FUNCTION_BLOCK "BFT_Garlic"   // FB362, LAD
{ S7_Optimized_Access := 'TRUE' }
VERSION : 0.1
// stored: AutoNumber false, IsIECCheckEnabled false, IsRetainMemResEnabled false, MemoryReserve 100, SetENOAutomatically false, UDAEnableTagReadback false
   VAR_INPUT
      IN_FBAV_Inload : Bool;
      IN_FBAV_Outlet : Bool;
      IN_FBAV_Transfer : Bool;
      IN_FBAV_CIP_Tank : Bool;
      IN_FBAV_CIP_Line : Bool;
      IN_FBP_Inload : Bool;
      IN_FBP_Inload_SP : Real;
      IN_FBP_Transfer : Bool;
      IN_FBP_Transfer_SP : Real;
      IN_FBP_CIP : Bool;
      IN_FBP_CIP_Sp : Real;
      IN_LT01 : Real;
      "LCS Start" : Bool;
      "LCS Stop" : Bool;
      "LCS EMS" : Bool;
      IN_Dose_Run : Bool;
      IN_Dose_Held : Bool;
      IN_Dose_Complete : Bool;
      IN_Dose_Header_1 : Bool;
      IN_Dose_Header_2 : Bool;
      IN_Dose_Valve_Cmd : Bool;
      IN_Dose_Pump_Cmd : Bool;
      IN_Dose_Pump_Sp : Real;
      IN_Dose_LineOK : Bool;
      "Inload Busy" : Bool;
      "CIP Pulse" : Bool;
      "CIP Supply ON" : Bool;
      "CIP Req OK" : Bool;
      "CIP Complete" : Bool;
      "CIP Busy" : Bool;
   END_VAR
   VAR_OUTPUT
      Out_AV_Inload : Bool;
      Out_AV_Outlet : Bool;
      Out_AV_Transfer : Bool;
      Out_AV_CIP_Tank : Bool;
      Out_AV_CIP_Line : Bool;
      Out_P_Inload : Bool;
      Out_P_Inload_Sp : Real;
      Out_P_Transfer : Bool;
      Out_P_Transfer_Sp : Real;
      Out_P_CIP : Bool;
      Out_P_CIP_Sp : Real;
      Out_XA : Bool;
      Out_XA_Speed : Real;
      Out_CIP_Req : Bool;
      Out_CIP_LineOpen : Bool;
   END_VAR
   VAR
      Cmd : Struct
         Inload : Bool;
         Ready_for_Tranfer : Bool;
         CIP_Tank : Bool;
         CIP_Line : Bool;
         Agitator_SpeedMode : Bool;
         Agitator_Mode : Bool;
         Agitator_Man_OnOff : Bool;
      END_STRUCT;
   END_VAR
   VAR RETAIN
      Param : Struct
         SP_Level_LL : Real := 10.0;
         SP_Level_ML : Real := 80.0;
         SP_Level_HL : Real := 100.0;
         SP_Level_Agi_ON1 : Real := 20.0;
         SP_Level_Agi_OFF1 : Real := 60.0;
         SP_Level_Agi_ON2 : Real := 62.0;
         SP_Level_Agi_OFF2 : Real := 80.0;
         SP_Level_Agi_ON3 : Real := 82.0;
         Agitator_SP_Speed : Real := 50.0;
         SupplyPump_SP_Speed : Real := 80.0;
         L_Hi_Lim : Real := 100.0;
         L_Lo_Lim : Real := 0.0;
         L_Hys : Real := 2.0;
         FlushingTime : DInt := 10000;
         CIP_Trf_SP_Speed : Real := 80.0;
         CIP_Ret_ON_SP : Real := 5.0;
         CIP_Ret_OFF_SP : Real;
      END_STRUCT;
   END_VAR
   VAR
      State : Struct   // Tank in loading state
         Tank_LL : Bool;
         Tank_ML : Bool;
         Tank_HL : Bool;
         Tank_inCIP : Bool;
         Tank_CIP_Enable : Bool;
         Line_inCIP : Bool;
         Line_CIP_Enable : Bool;
         CIP_Return_On : Bool;
         Inloading : Bool;
         Inload_Enable : Bool;
         Ready_For_Transfer : Bool;
         Ready_For_Transfer_Ena : Bool;
         Tank_Available : Bool;
         Transfer_On_Prog : Bool;
         L_Agi_ON1 : Bool;
         L_Agi_ON2 : Bool;
         L_Agi_ON3 : Bool;
      END_STRUCT;
      alwaysON : Bool;
      L_Hys_Abs : Real;
      Hys_Level_HL : Real;
      Hys_Level_ML : Real;
      Hys_Level_LL : Real;
      Hys_Level_Agi : Real;
      r : Struct
         PosE1 : Bool;
         PosE2 : Bool;
         PosE3 : Bool;
         PosE4 : Bool;
         PosE5 : Bool;
         PosE6 : Bool;
         PosE7 : Bool;
         PosE8 : Bool;
         PosE9 : Bool;
         PosE10 : Bool;
         PosE11 : Bool;
         PosE12 : Bool;
         PosE13 : Bool;
         PosE14 : Bool;
         PosE15 : Bool;
         PosE16 : Bool;
         PosE17 : Bool;
         PosE18 : Bool;
         PosE19 : Bool;
         PosE20 : Bool;
         PosE21 : Bool;
         PosE22 : Bool;
         PosE23 : Bool;
         PosE24 : Bool;
         PosE25 : Bool;
         PosE26 : Bool;
         PosE27 : Bool;
         PosE28 : Bool;
         PosE29 : Bool;
         PosE30 : Bool;
         PosE31 : Bool;
         PosE32 : Bool;
      END_STRUCT;
      Actuator : Struct
         AV_Inload : Bool;
         AV_Outlet : Bool;
         AV_Transfer : Bool;
         AV_CIP_Tank : Bool;
         AV_CIP_Line : Bool;
         P_Transfer : Bool;
         P_Inload : Bool;
         P_CIP : Bool;
         Agitator_level : Bool;
         LCS_OnOff : Bool;
      END_STRUCT;
      FlushingTim : TON_TIME;
      SPumpTim { S7_SetPoint := 'True'} : TON_TIME;
      AVinloadTim { S7_SetPoint := 'True'} : TON_TIME;
      L_AgiTim { S7_SetPoint := 'True'} : TON_TIME;
      Pump_TF_On_Time { S7_SetPoint := 'True'} : TON_TIME;
   END_VAR
   VAR_TEMP   // added for the SCL form of the ladder/FBD networks
      _w1 : Bool;
      _w2 : Bool;
   END_VAR
BEGIN

REGION Network 1: Always_ON
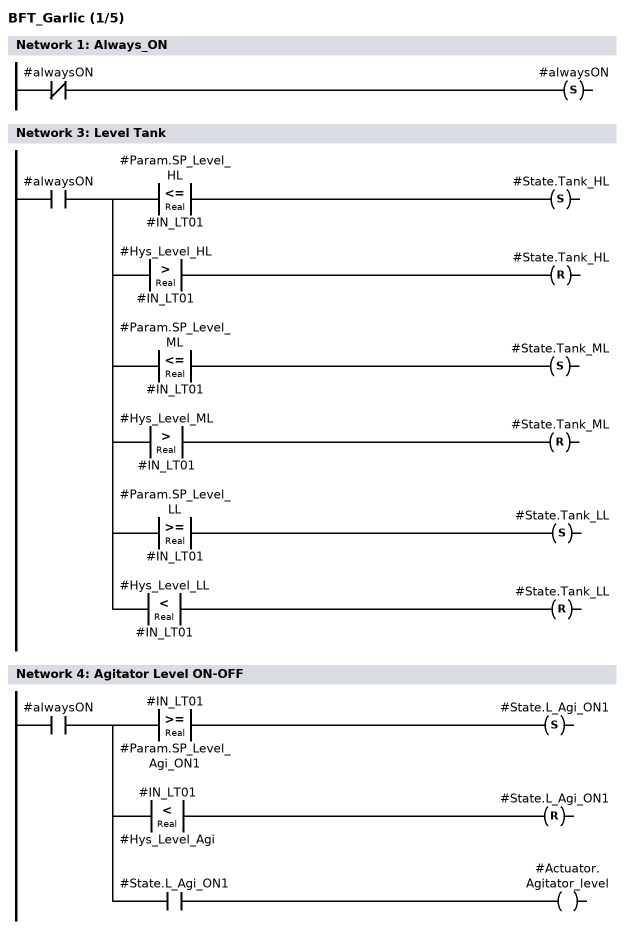
   RUNG wire#powerrail
      I_Contact( #alwaysON )
      S_Coil( #alwaysON )
   END_RUNG
   // the same network as SCL:
   IF NOT #alwaysON THEN #alwaysON := TRUE; END_IF;
END_REGION

NETWORK
TITLE = Hys Calculation
//Level Hys Absolute
      L     #Param.L_Hi_Lim;
      L     #Param.L_Lo_Lim;
      -R;
      L     100.0;
      /R;
      L     #Param.L_Hys;
      *R;
      T     #L_Hys_Abs;
//Tank High Level
      L     #Param.SP_Level_HL;
      L     #L_Hys_Abs;
      -R;
      T     #Hys_Level_HL;
//Tank Mid Level
      L     #Param.SP_Level_ML;
      L     #L_Hys_Abs;
      -R;
      T     #Hys_Level_ML;
//Tank Low Level
      L     #Param.SP_Level_LL;
      L     #L_Hys_Abs;
      +R;
      T     #Hys_Level_LL;
//Level Agi
      L     #Param.SP_Level_Agi_ON1;
      L     #L_Hys_Abs;
      -R;
      T     #Hys_Level_Agi;



REGION Network 3: Level Tank
   RUNG wire#powerrail
      Contact( #alwaysON )
      wire#w1
      { S7_Templates := "SrcType := Real" } LE_Contact(in1 := #Param.SP_Level_HL, in2 := #IN_LT01)
      S_Coil( #State.Tank_HL )
   END_RUNG
   RUNG wire#w1
      { S7_Templates := "SrcType := Real" } GT_Contact(in1 := #Hys_Level_HL, in2 := #IN_LT01)
      R_Coil( #State.Tank_HL )
   END_RUNG
   RUNG wire#w1
      { S7_Templates := "SrcType := Real" } LE_Contact(in1 := #Param.SP_Level_ML, in2 := #IN_LT01)
      S_Coil( #State.Tank_ML )
   END_RUNG
   RUNG wire#w1
      { S7_Templates := "SrcType := Real" } GT_Contact(in1 := #Hys_Level_ML, in2 := #IN_LT01)
      R_Coil( #State.Tank_ML )
   END_RUNG
   RUNG wire#w1
      { S7_Templates := "SrcType := Real" } GE_Contact(in1 := #Param.SP_Level_LL, in2 := #IN_LT01)
      S_Coil( #State.Tank_LL )
   END_RUNG
   RUNG wire#w1
      { S7_Templates := "SrcType := Real" } LT_Contact(in1 := #Hys_Level_LL, in2 := #IN_LT01)
      R_Coil( #State.Tank_LL )
   END_RUNG
   // the same network as SCL:
   IF #alwaysON AND (#Param.SP_Level_HL <= #IN_LT01) THEN #State.Tank_HL := TRUE; END_IF;
   IF #alwaysON AND (#Hys_Level_HL > #IN_LT01) THEN #State.Tank_HL := FALSE; END_IF;
   IF #alwaysON AND (#Param.SP_Level_ML <= #IN_LT01) THEN #State.Tank_ML := TRUE; END_IF;
   IF #alwaysON AND (#Hys_Level_ML > #IN_LT01) THEN #State.Tank_ML := FALSE; END_IF;
   IF #alwaysON AND (#Param.SP_Level_LL >= #IN_LT01) THEN #State.Tank_LL := TRUE; END_IF;
   IF #alwaysON AND (#Hys_Level_LL < #IN_LT01) THEN #State.Tank_LL := FALSE; END_IF;
END_REGION

REGION Network 4: Agitator Level ON-OFF
   RUNG wire#powerrail
      Contact( #alwaysON )
      wire#w1
      { S7_Templates := "SrcType := Real" } GE_Contact(in1 := #IN_LT01, in2 := #Param.SP_Level_Agi_ON1)
      S_Coil( #State.L_Agi_ON1 )
   END_RUNG
   RUNG wire#w1
      { S7_Templates := "SrcType := Real" } LT_Contact(in1 := #IN_LT01, in2 := #Hys_Level_Agi)
      R_Coil( #State.L_Agi_ON1 )
   END_RUNG
   RUNG wire#w1
      Contact( #State.L_Agi_ON1 )
      Coil( #Actuator.Agitator_level )
   END_RUNG
   // the same network as SCL:
   IF #alwaysON AND (#IN_LT01 >= #Param.SP_Level_Agi_ON1) THEN #State.L_Agi_ON1 := TRUE; END_IF;
   IF #alwaysON AND (#IN_LT01 < #Hys_Level_Agi) THEN #State.L_Agi_ON1 := FALSE; END_IF;
   #Actuator.Agitator_level := #alwaysON AND #State.L_Agi_ON1;
END_REGION

REGION Network 5: Agitator
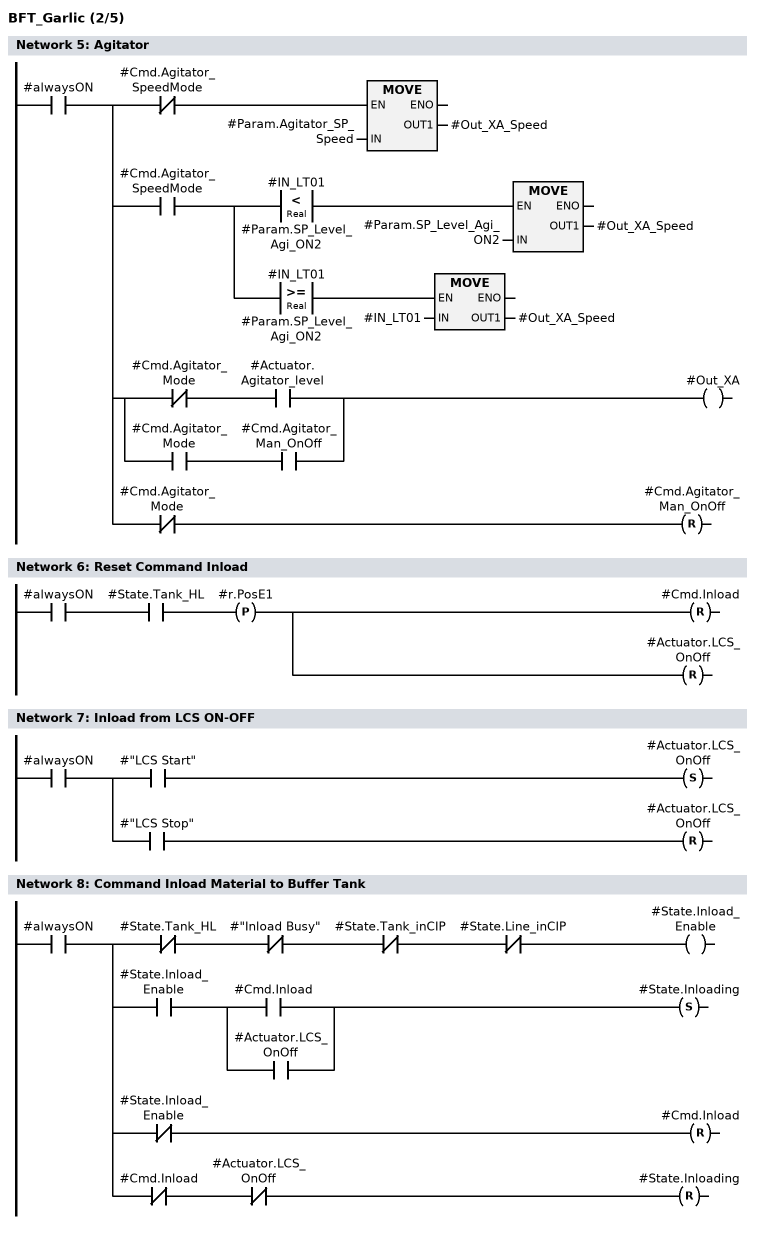
   RUNG wire#powerrail
      Contact( #alwaysON )
      wire#w1
      I_Contact( #Cmd.Agitator_SpeedMode )
      Move(in := #Param.Agitator_SP_Speed, out1 => #Out_XA_Speed)
   END_RUNG
   RUNG wire#w1
      Contact( #Cmd.Agitator_SpeedMode )
      wire#w2
      { S7_Templates := "SrcType := Real" } LT_Contact(in1 := #IN_LT01, in2 := #Param.SP_Level_Agi_ON2)
      Move(in := #Param.SP_Level_Agi_ON2, out1 => #Out_XA_Speed)
   END_RUNG
   RUNG wire#w2
      { S7_Templates := "SrcType := Real" } GE_Contact(in1 := #IN_LT01, in2 := #Param.SP_Level_Agi_ON2)
      Move(in := #IN_LT01, out1 => #Out_XA_Speed)
   END_RUNG
   RUNG wire#w1
      I_Contact( #Cmd.Agitator_Mode )
      Contact( #Actuator.Agitator_level )
      wire#w3
      Coil( #Out_XA )
   END_RUNG
   RUNG wire#w1
      Contact( #Cmd.Agitator_Mode )
      Contact( #Cmd.Agitator_Man_OnOff )
   END_RUNG wire#w3
   RUNG wire#w1
      I_Contact( #Cmd.Agitator_Mode )
      R_Coil( #Cmd.Agitator_Man_OnOff )
   END_RUNG
   // the same network as SCL:
   IF #alwaysON AND NOT #Cmd.Agitator_SpeedMode THEN #Out_XA_Speed := #Param.Agitator_SP_Speed; END_IF;
   #_w1 := #alwaysON AND #Cmd.Agitator_SpeedMode;
   IF #_w1 AND (#IN_LT01 < #Param.SP_Level_Agi_ON2) THEN #Out_XA_Speed := #Param.SP_Level_Agi_ON2; END_IF;
   IF #_w1 AND (#IN_LT01 >= #Param.SP_Level_Agi_ON2) THEN #Out_XA_Speed := #IN_LT01; END_IF;
   #Out_XA := #alwaysON AND ((NOT #Cmd.Agitator_Mode AND #Actuator.Agitator_level) OR (#Cmd.Agitator_Mode AND #Cmd.Agitator_Man_OnOff));
   IF #alwaysON AND NOT #Cmd.Agitator_Mode THEN #Cmd.Agitator_Man_OnOff := FALSE; END_IF;
END_REGION

REGION Network 6: Reset Command Inload
   RUNG wire#powerrail
      Contact( #alwaysON )
      Contact( #State.Tank_HL )
      P_Trig( #r.PosE1 )
      wire#w1
      R_Coil( #Cmd.Inload )
   END_RUNG
   RUNG wire#w1
      R_Coil( #Actuator.LCS_OnOff )
   END_RUNG
   // the same network as SCL:
   #_w1 := #alwaysON AND #State.Tank_HL;
   #_w2 := #_w1 AND NOT #r.PosE1;   // rising edge
   #r.PosE1 := #_w1;
   IF #_w2 THEN
       #Cmd.Inload := FALSE;
       #Actuator.LCS_OnOff := FALSE;
   END_IF;
END_REGION

REGION Network 7: Inload from LCS ON-OFF
   RUNG wire#powerrail
      Contact( #alwaysON )
      wire#w1
      Contact( #"LCS Start" )
      S_Coil( #Actuator.LCS_OnOff )
   END_RUNG
   RUNG wire#w1
      Contact( #"LCS Stop" )
      R_Coil( #Actuator.LCS_OnOff )
   END_RUNG
   // the same network as SCL:
   IF #alwaysON AND #"LCS Start" THEN #Actuator.LCS_OnOff := TRUE; END_IF;
   IF #alwaysON AND #"LCS Stop" THEN #Actuator.LCS_OnOff := FALSE; END_IF;
END_REGION

REGION Network 8: Command Inload Material to Buffer Tank
   RUNG wire#powerrail
      Contact( #alwaysON )
      wire#w1
      I_Contact( #State.Tank_HL )
      I_Contact( #"Inload Busy" )
      I_Contact( #State.Tank_inCIP )
      I_Contact( #State.Line_inCIP )
      Coil( #State.Inload_Enable )
   END_RUNG
   RUNG wire#w1
      Contact( #State.Inload_Enable )
      wire#w2
      Contact( #Cmd.Inload )
      wire#w3
      S_Coil( #State.Inloading )
   END_RUNG
   RUNG wire#w2
      Contact( #Actuator.LCS_OnOff )
   END_RUNG wire#w3
   RUNG wire#w1
      I_Contact( #State.Inload_Enable )
      R_Coil( #Cmd.Inload )
   END_RUNG
   RUNG wire#w1
      I_Contact( #Cmd.Inload )
      I_Contact( #Actuator.LCS_OnOff )
      R_Coil( #State.Inloading )
   END_RUNG
   // the same network as SCL:
   #State.Inload_Enable := #alwaysON AND NOT #State.Tank_HL AND NOT #"Inload Busy" AND NOT #State.Tank_inCIP AND NOT #State.Line_inCIP;
   IF #alwaysON AND #State.Inload_Enable AND (#Cmd.Inload OR #Actuator.LCS_OnOff) THEN
       #State.Inloading := TRUE;
   END_IF;
   IF #alwaysON AND NOT #State.Inload_Enable THEN #Cmd.Inload := FALSE; END_IF;
   IF #alwaysON AND NOT #Cmd.Inload AND NOT #Actuator.LCS_OnOff THEN #State.Inloading := FALSE; END_IF;
END_REGION

REGION Network 9: Tank Ready for Transfer to Blending
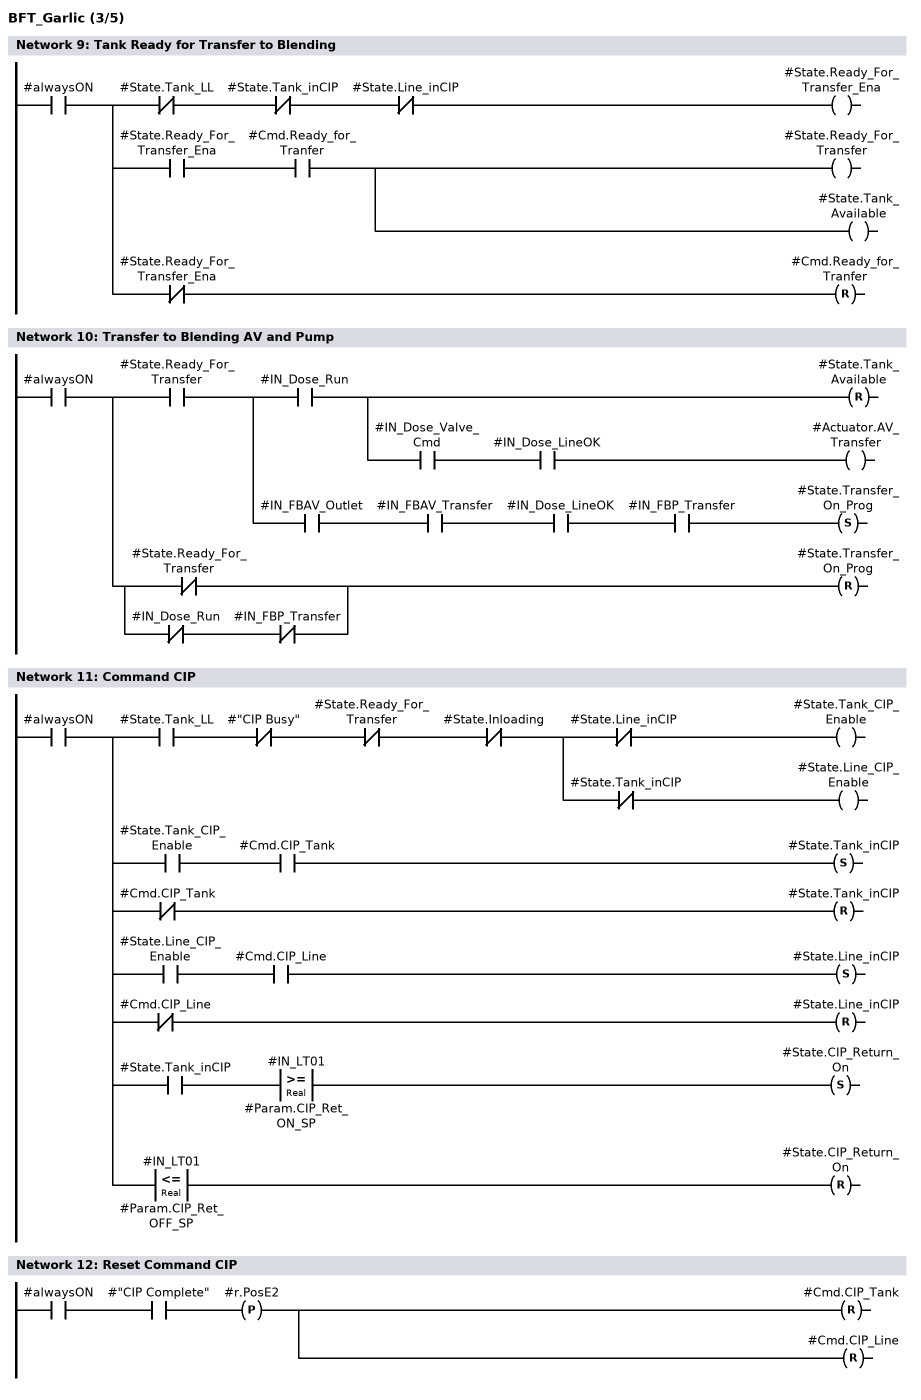
   RUNG wire#powerrail
      Contact( #alwaysON )
      wire#w1
      I_Contact( #State.Tank_LL )
      I_Contact( #State.Tank_inCIP )
      I_Contact( #State.Line_inCIP )
      Coil( #State.Ready_For_Transfer_Ena )
   END_RUNG
   RUNG wire#w1
      Contact( #State.Ready_For_Transfer_Ena )
      Contact( #Cmd.Ready_for_Tranfer )
      wire#w2
      Coil( #State.Ready_For_Transfer )
   END_RUNG
   RUNG wire#w2
      Coil( #State.Tank_Available )
   END_RUNG
   RUNG wire#w1
      I_Contact( #State.Ready_For_Transfer_Ena )
      R_Coil( #Cmd.Ready_for_Tranfer )
   END_RUNG
   // the same network as SCL:
   #State.Ready_For_Transfer_Ena := #alwaysON AND NOT #State.Tank_LL AND NOT #State.Tank_inCIP AND NOT #State.Line_inCIP;
   #State.Ready_For_Transfer := #alwaysON AND #State.Ready_For_Transfer_Ena AND #Cmd.Ready_for_Tranfer;
   #State.Tank_Available := #State.Ready_For_Transfer;
   IF #alwaysON AND NOT #State.Ready_For_Transfer_Ena THEN #Cmd.Ready_for_Tranfer := FALSE; END_IF;
END_REGION

REGION Network 10: Transfer to Blending AV and Pump
   RUNG wire#powerrail
      Contact( #alwaysON )
      wire#w1
      Contact( #State.Ready_For_Transfer )
      wire#w2
      Contact( #IN_Dose_Run )
      wire#w3
      R_Coil( #State.Tank_Available )
   END_RUNG
   RUNG wire#w3
      Contact( #IN_Dose_Valve_Cmd )
      Contact( #IN_Dose_LineOK )
      Coil( #Actuator.AV_Transfer )
   END_RUNG
   RUNG wire#w2
      Contact( #IN_FBAV_Outlet )
      Contact( #IN_FBAV_Transfer )
      Contact( #IN_Dose_LineOK )
      Contact( #IN_FBP_Transfer )
      S_Coil( #State.Transfer_On_Prog )
   END_RUNG
   RUNG wire#w1
      I_Contact( #State.Ready_For_Transfer )
      wire#w4
      R_Coil( #State.Transfer_On_Prog )
   END_RUNG
   RUNG wire#w1
      I_Contact( #IN_Dose_Run )
      I_Contact( #IN_FBP_Transfer )
   END_RUNG wire#w4
   // the same network as SCL:
   #_w1 := #alwaysON AND #State.Ready_For_Transfer;
   #_w2 := #_w1 AND #IN_Dose_Run;
   IF #_w2 THEN #State.Tank_Available := FALSE; END_IF;
   #Actuator.AV_Transfer := #_w2 AND #IN_Dose_Valve_Cmd AND #IN_Dose_LineOK;
   IF #_w1 AND #IN_FBAV_Outlet AND #IN_FBAV_Transfer AND #IN_Dose_LineOK AND #IN_FBP_Transfer THEN
       #State.Transfer_On_Prog := TRUE;
   END_IF;
   IF #alwaysON AND (NOT #State.Ready_For_Transfer OR (NOT #IN_Dose_Run AND NOT #IN_FBP_Transfer)) THEN
       #State.Transfer_On_Prog := FALSE;
   END_IF;
END_REGION

REGION Network 11: Command CIP
   RUNG wire#powerrail
      Contact( #alwaysON )
      wire#w1
      Contact( #State.Tank_LL )
      I_Contact( #"CIP Busy" )
      I_Contact( #State.Ready_For_Transfer )
      I_Contact( #State.Inloading )
      wire#w2
      I_Contact( #State.Line_inCIP )
      Coil( #State.Tank_CIP_Enable )
   END_RUNG
   RUNG wire#w2
      I_Contact( #State.Tank_inCIP )
      Coil( #State.Line_CIP_Enable )
   END_RUNG
   RUNG wire#w1
      Contact( #State.Tank_CIP_Enable )
      Contact( #Cmd.CIP_Tank )
      S_Coil( #State.Tank_inCIP )
   END_RUNG
   RUNG wire#w1
      I_Contact( #Cmd.CIP_Tank )
      R_Coil( #State.Tank_inCIP )
   END_RUNG
   RUNG wire#w1
      Contact( #State.Line_CIP_Enable )
      Contact( #Cmd.CIP_Line )
      S_Coil( #State.Line_inCIP )
   END_RUNG
   RUNG wire#w1
      I_Contact( #Cmd.CIP_Line )
      R_Coil( #State.Line_inCIP )
   END_RUNG
   RUNG wire#w1
      Contact( #State.Tank_inCIP )
      { S7_Templates := "SrcType := Real" } GE_Contact(in1 := #IN_LT01, in2 := #Param.CIP_Ret_ON_SP)
      S_Coil( #State.CIP_Return_On )
   END_RUNG
   RUNG wire#w1
      { S7_Templates := "SrcType := Real" } LE_Contact(in1 := #IN_LT01, in2 := #Param.CIP_Ret_OFF_SP)
      R_Coil( #State.CIP_Return_On )
   END_RUNG
   // the same network as SCL:
   #_w1 := #alwaysON AND #State.Tank_LL AND NOT #"CIP Busy" AND NOT #State.Ready_For_Transfer AND NOT #State.Inloading;
   #State.Tank_CIP_Enable := #_w1 AND NOT #State.Line_inCIP;
   #State.Line_CIP_Enable := #_w1 AND NOT #State.Tank_inCIP;
   IF #alwaysON AND #State.Tank_CIP_Enable AND #Cmd.CIP_Tank THEN #State.Tank_inCIP := TRUE; END_IF;
   IF #alwaysON AND NOT #Cmd.CIP_Tank THEN #State.Tank_inCIP := FALSE; END_IF;
   IF #alwaysON AND #State.Line_CIP_Enable AND #Cmd.CIP_Line THEN #State.Line_inCIP := TRUE; END_IF;
   IF #alwaysON AND NOT #Cmd.CIP_Line THEN #State.Line_inCIP := FALSE; END_IF;
   IF #alwaysON AND #State.Tank_inCIP AND (#IN_LT01 >= #Param.CIP_Ret_ON_SP) THEN
       #State.CIP_Return_On := TRUE;
   END_IF;
   IF #alwaysON AND (#IN_LT01 <= #Param.CIP_Ret_OFF_SP) THEN #State.CIP_Return_On := FALSE; END_IF;
END_REGION

REGION Network 12: Reset Command CIP
   RUNG wire#powerrail
      Contact( #alwaysON )
      Contact( #"CIP Complete" )
      P_Trig( #r.PosE2 )
      wire#w1
      R_Coil( #Cmd.CIP_Tank )
   END_RUNG
   RUNG wire#w1
      R_Coil( #Cmd.CIP_Line )
   END_RUNG
   // the same network as SCL:
   #_w1 := #alwaysON AND #"CIP Complete";
   #_w2 := #_w1 AND NOT #r.PosE2;   // rising edge
   #r.PosE2 := #_w1;
   IF #_w2 THEN
       #Cmd.CIP_Tank := FALSE;
       #Cmd.CIP_Line := FALSE;
   END_IF;
END_REGION

REGION Network 13: CIP Request and CIP Line Open
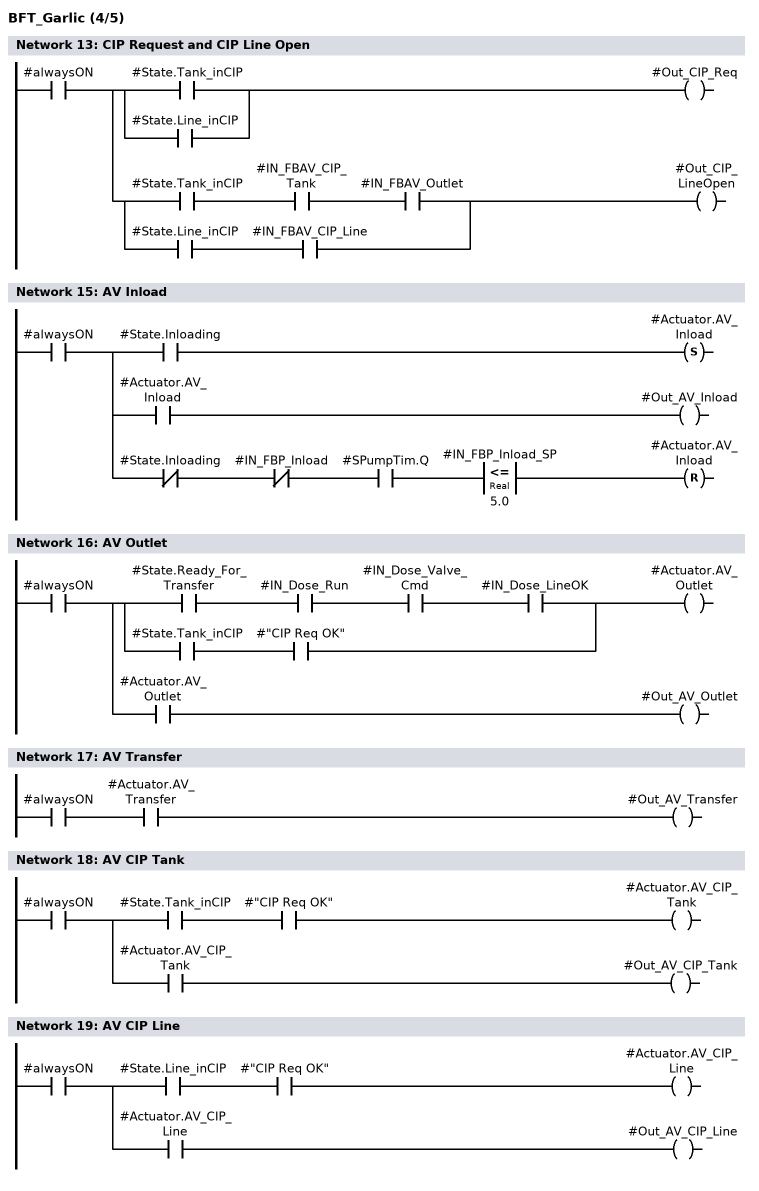
   RUNG wire#powerrail
      Contact( #alwaysON )
      wire#w1
      Contact( #State.Tank_inCIP )
      wire#w2
      Coil( #Out_CIP_Req )
   END_RUNG
   RUNG wire#w1
      Contact( #State.Line_inCIP )
   END_RUNG wire#w2
   RUNG wire#w1
      Contact( #State.Tank_inCIP )
      Contact( #IN_FBAV_CIP_Tank )
      Contact( #IN_FBAV_Outlet )
      wire#w3
      Coil( #Out_CIP_LineOpen )
   END_RUNG
   RUNG wire#w1
      Contact( #State.Line_inCIP )
      Contact( #IN_FBAV_CIP_Line )
   END_RUNG wire#w3
   // the same network as SCL:
   #Out_CIP_Req := #alwaysON AND (#State.Tank_inCIP OR #State.Line_inCIP);
   #Out_CIP_LineOpen := #alwaysON AND ((#State.Tank_inCIP AND #IN_FBAV_CIP_Tank AND #IN_FBAV_Outlet) OR (#State.Line_inCIP AND #IN_FBAV_CIP_Line));
END_REGION

REGION Network 15: AV Inload
   RUNG wire#powerrail
      Contact( #alwaysON )
      wire#w1
      Contact( #State.Inloading )
      S_Coil( #Actuator.AV_Inload )
   END_RUNG
   RUNG wire#w1
      Contact( #Actuator.AV_Inload )
      Coil( #Out_AV_Inload )
   END_RUNG
   RUNG wire#w1
      I_Contact( #State.Inloading )
      I_Contact( #IN_FBP_Inload )
      Contact( #SPumpTim.Q )
      { S7_Templates := "SrcType := Real" } LE_Contact(in1 := #IN_FBP_Inload_SP, in2 := 5.0)
      R_Coil( #Actuator.AV_Inload )
   END_RUNG
   // the same network as SCL:
   IF #alwaysON AND #State.Inloading THEN #Actuator.AV_Inload := TRUE; END_IF;
   #Out_AV_Inload := #alwaysON AND #Actuator.AV_Inload;
   IF #alwaysON AND NOT #State.Inloading AND NOT #IN_FBP_Inload AND #SPumpTim.Q AND (#IN_FBP_Inload_SP <= 5.0) THEN
       #Actuator.AV_Inload := FALSE;
   END_IF;
END_REGION

REGION Network 16: AV Outlet
   RUNG wire#powerrail
      Contact( #alwaysON )
      wire#w1
      Contact( #State.Ready_For_Transfer )
      Contact( #IN_Dose_Run )
      Contact( #IN_Dose_Valve_Cmd )
      Contact( #IN_Dose_LineOK )
      wire#w2
      Coil( #Actuator.AV_Outlet )
   END_RUNG
   RUNG wire#w1
      Contact( #State.Tank_inCIP )
      Contact( #"CIP Req OK" )
   END_RUNG wire#w2
   RUNG wire#w1
      Contact( #Actuator.AV_Outlet )
      Coil( #Out_AV_Outlet )
   END_RUNG
   // the same network as SCL:
   #Actuator.AV_Outlet := #alwaysON AND ((#State.Ready_For_Transfer AND #IN_Dose_Run AND #IN_Dose_Valve_Cmd AND #IN_Dose_LineOK) OR (#State.Tank_inCIP AND #"CIP Req OK"));
   #Out_AV_Outlet := #alwaysON AND #Actuator.AV_Outlet;
END_REGION

REGION Network 17: AV Transfer
   RUNG wire#powerrail
      Contact( #alwaysON )
      Contact( #Actuator.AV_Transfer )
      Coil( #Out_AV_Transfer )
   END_RUNG
   // the same network as SCL:
   #Out_AV_Transfer := #alwaysON AND #Actuator.AV_Transfer;
END_REGION

REGION Network 18: AV CIP Tank
   RUNG wire#powerrail
      Contact( #alwaysON )
      wire#w1
      Contact( #State.Tank_inCIP )
      Contact( #"CIP Req OK" )
      Coil( #Actuator.AV_CIP_Tank )
   END_RUNG
   RUNG wire#w1
      Contact( #Actuator.AV_CIP_Tank )
      Coil( #Out_AV_CIP_Tank )
   END_RUNG
   // the same network as SCL:
   #Actuator.AV_CIP_Tank := #alwaysON AND #State.Tank_inCIP AND #"CIP Req OK";
   #Out_AV_CIP_Tank := #alwaysON AND #Actuator.AV_CIP_Tank;
END_REGION

REGION Network 19: AV CIP Line
   RUNG wire#powerrail
      Contact( #alwaysON )
      wire#w1
      Contact( #State.Line_inCIP )
      Contact( #"CIP Req OK" )
      Coil( #Actuator.AV_CIP_Line )
   END_RUNG
   RUNG wire#w1
      Contact( #Actuator.AV_CIP_Line )
      Coil( #Out_AV_CIP_Line )
   END_RUNG
   // the same network as SCL:
   #Actuator.AV_CIP_Line := #alwaysON AND #State.Line_inCIP AND #"CIP Req OK";
   #Out_AV_CIP_Line := #alwaysON AND #Actuator.AV_CIP_Line;
END_REGION

REGION Network 21: Pump Inload
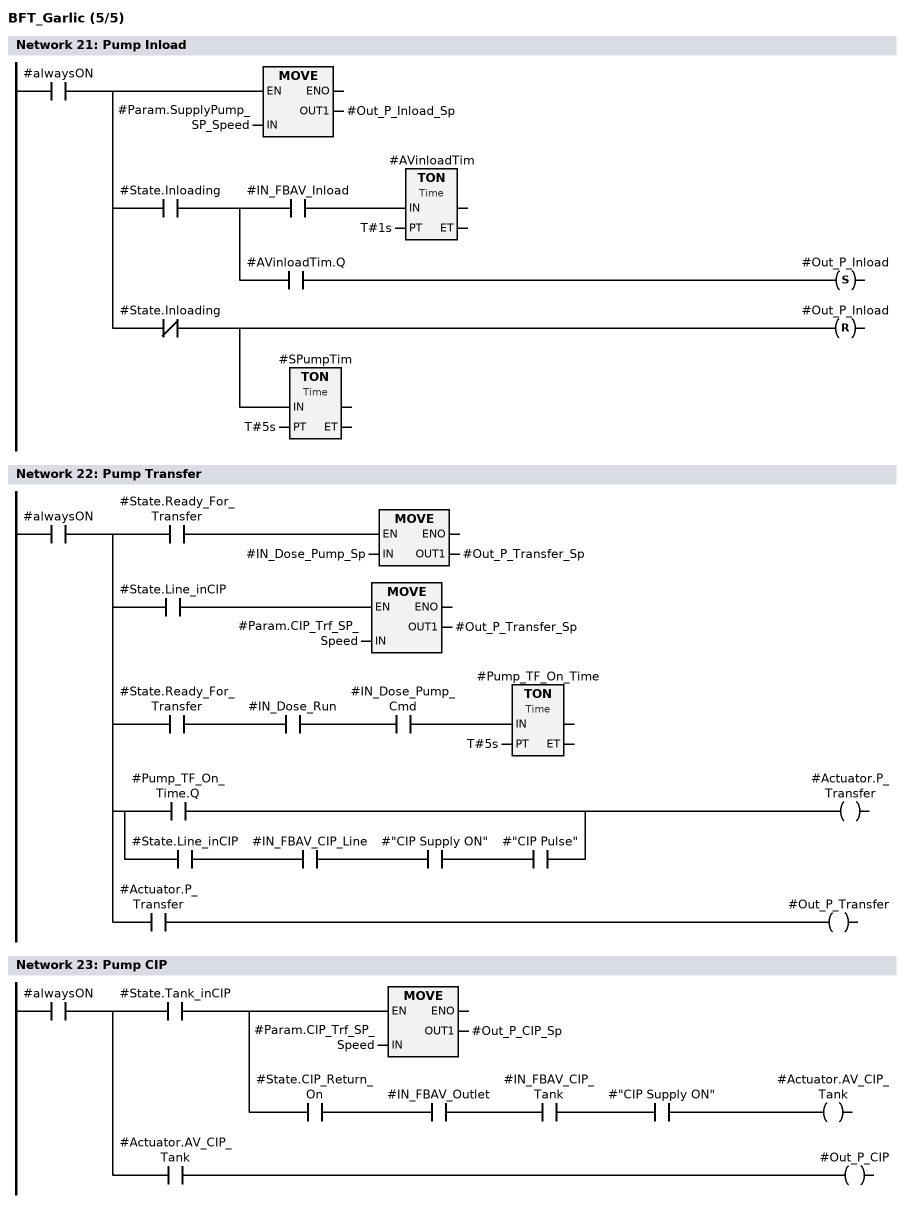
   RUNG wire#powerrail
      Contact( #alwaysON )
      wire#w1
      Move(in := #Param.SupplyPump_SP_Speed, out1 => #Out_P_Inload_Sp)
   END_RUNG
   RUNG wire#w1
      Contact( #State.Inloading )
      wire#w2
      Contact( #IN_FBAV_Inload )
      { S7_Templates := "time_type := Time" } #AVinloadTim.TON(pt := T#1s, et =>)
   END_RUNG
   RUNG wire#w2
      Contact( #AVinloadTim.Q )
      S_Coil( #Out_P_Inload )
   END_RUNG
   RUNG wire#w1
      I_Contact( #State.Inloading )
      wire#w3
      R_Coil( #Out_P_Inload )
   END_RUNG
   RUNG wire#w3
      { S7_Templates := "time_type := Time" } #SPumpTim.TON(pt := T#5s, et =>)
   END_RUNG
   // the same network as SCL:
   IF #alwaysON THEN #Out_P_Inload_Sp := #Param.SupplyPump_SP_Speed; END_IF;
   #_w1 := #alwaysON AND #State.Inloading;
   #AVinloadTim(IN := #_w1 AND #IN_FBAV_Inload, PT := T#1s);   // TON
   IF #_w1 AND #AVinloadTim.Q THEN #Out_P_Inload := TRUE; END_IF;
   #_w2 := #alwaysON AND NOT #State.Inloading;
   IF #_w2 THEN #Out_P_Inload := FALSE; END_IF;
   #SPumpTim(IN := #_w2, PT := T#5s);   // TON
END_REGION

REGION Network 22: Pump Transfer
   RUNG wire#powerrail
      Contact( #alwaysON )
      wire#w1
      Contact( #State.Ready_For_Transfer )
      Move(in := #IN_Dose_Pump_Sp, out1 => #Out_P_Transfer_Sp)
   END_RUNG
   RUNG wire#w1
      Contact( #State.Line_inCIP )
      Move(in := #Param.CIP_Trf_SP_Speed, out1 => #Out_P_Transfer_Sp)
   END_RUNG
   RUNG wire#w1
      Contact( #State.Ready_For_Transfer )
      Contact( #IN_Dose_Run )
      Contact( #IN_Dose_Pump_Cmd )
      { S7_Templates := "time_type := Time" } #Pump_TF_On_Time.TON(pt := T#5s, et =>)
   END_RUNG
   RUNG wire#w1
      Contact( #Pump_TF_On_Time.Q )
      wire#w2
      Coil( #Actuator.P_Transfer )
   END_RUNG
   RUNG wire#w1
      Contact( #State.Line_inCIP )
      Contact( #IN_FBAV_CIP_Line )
      Contact( #"CIP Supply ON" )
      Contact( #"CIP Pulse" )
   END_RUNG wire#w2
   RUNG wire#w1
      Contact( #Actuator.P_Transfer )
      Coil( #Out_P_Transfer )
   END_RUNG
   // the same network as SCL:
   IF #alwaysON AND #State.Ready_For_Transfer THEN #Out_P_Transfer_Sp := #IN_Dose_Pump_Sp; END_IF;
   IF #alwaysON AND #State.Line_inCIP THEN #Out_P_Transfer_Sp := #Param.CIP_Trf_SP_Speed; END_IF;
   #Pump_TF_On_Time(IN := #alwaysON AND #State.Ready_For_Transfer AND #IN_Dose_Run AND #IN_Dose_Pump_Cmd,   // TON
                    PT := T#5s);
   #Actuator.P_Transfer := #alwaysON AND (#Pump_TF_On_Time.Q OR (#State.Line_inCIP AND #IN_FBAV_CIP_Line AND #"CIP Supply ON" AND #"CIP Pulse"));
   #Out_P_Transfer := #alwaysON AND #Actuator.P_Transfer;
END_REGION

REGION Network 23: Pump CIP
   RUNG wire#powerrail
      Contact( #alwaysON )
      wire#w1
      Contact( #State.Tank_inCIP )
      wire#w2
      Move(in := #Param.CIP_Trf_SP_Speed, out1 => #Out_P_CIP_Sp)
   END_RUNG
   RUNG wire#w2
      Contact( #State.CIP_Return_On )
      Contact( #IN_FBAV_Outlet )
      Contact( #IN_FBAV_CIP_Tank )
      Contact( #"CIP Supply ON" )
      Coil( #Actuator.AV_CIP_Tank )
   END_RUNG
   RUNG wire#w1
      Contact( #Actuator.AV_CIP_Tank )
      Coil( #Out_P_CIP )
   END_RUNG
   // the same network as SCL:
   #_w1 := #alwaysON AND #State.Tank_inCIP;
   IF #_w1 THEN #Out_P_CIP_Sp := #Param.CIP_Trf_SP_Speed; END_IF;
   #Actuator.AV_CIP_Tank := #_w1 AND #State.CIP_Return_On AND #IN_FBAV_Outlet AND #IN_FBAV_CIP_Tank AND #"CIP Supply ON";
   #Out_P_CIP := #alwaysON AND #Actuator.AV_CIP_Tank;
END_REGION
END_FUNCTION_BLOCK

FUNCTION_BLOCK "BFT_Vinegar"   // FB363, LAD
{ S7_Optimized_Access := 'TRUE' }
VERSION : 0.1
// stored: AutoNumber false, IsIECCheckEnabled false, IsRetainMemResEnabled false, MemoryReserve 100, SetENOAutomatically false, UDAEnableTagReadback false
   VAR_INPUT
      IN_FBAV_Inload : Bool;
      IN_FBAV_Outlet : Bool;
      IN_FBAV_Transfer : Bool;
      IN_FBAV_CIP_Tank : Bool;
      IN_FBAV_CIP_Line : Bool;
      IN_FBP_Inload : Bool;
      IN_FBP_Inload_SP : Real;
      IN_FBP_Transfer : Bool;
      IN_FBP_Transfer_SP : Real;
      IN_FBP_CIP : Bool;
      IN_FBP_CIP_Sp : Real;
      IN_LT01 : Real;
      "LCS Start" : Bool;
      "LCS Stop" : Bool;
      "LCS EMS" : Bool;
      IN_Dose_Run : Bool;
      IN_Dose_Held : Bool;
      IN_Dose_Complete : Bool;
      IN_Dose_Valve_Cmd : Bool;
      IN_Dose_Pump_Cmd : Bool;
      IN_Dose_Pump_Sp : Real;
      IN_Dose_LineOK : Bool;
      "Inload Busy" : Bool;
      "CIP Pulse" : Bool;
      "CIP Supply ON" : Bool;
      "CIP Req OK" : Bool;
      "CIP Complete" : Bool;
      "CIP Busy" : Bool;
   END_VAR
   VAR_OUTPUT
      Out_AV_Inload : Bool;
      Out_AV_Outlet : Bool;
      Out_AV_Transfer : Bool;
      Out_AV_CIP_Tank : Bool;
      Out_AV_CIP_Line : Bool;
      Out_P_Inload : Bool;
      Out_P_Inload_Sp : Real;
      Out_P_Transfer : Bool;
      Out_P_Transfer_Sp : Real;
      Out_P_CIP : Bool;
      Out_P_CIP_Sp : Real;
      Out_CIP_Req : Bool;
      Out_CIP_LineOpen : Bool;
   END_VAR
   VAR
      Cmd : Struct
         Inload : Bool;
         Ready_for_Tranfer : Bool;
         CIP_Tank : Bool;
         CIP_Line : Bool;
      END_STRUCT;
   END_VAR
   VAR RETAIN
      Param : Struct
         SP_Level_LL : Real := 10.0;
         SP_Level_ML : Real := 80.0;
         SP_Level_HL : Real := 100.0;
         SupplyPump_SP_Speed : Real := 80.0;
         L_Hi_Lim : Real := 100.0;
         L_Lo_Lim : Real := 0.0;
         L_Hys : Real := 2.0;
         FlushingTime : DInt := 10000;
         CIP_Trf_SP_Speed : Real := 80.0;
         CIP_Ret_ON_SP : Real := 5.0;
         CIP_Ret_OFF_SP : Real;
      END_STRUCT;
   END_VAR
   VAR
      State : Struct   // Tank in loading state
         Tank_LL : Bool;
         Tank_ML : Bool;
         Tank_HL : Bool;
         Tank_inCIP : Bool;
         Tank_CIP_Enable : Bool;
         Line_inCIP : Bool;
         Line_CIP_Enable : Bool;
         CIP_Return_On : Bool;
         Inloading : Bool;
         Inload_Enable : Bool;
         Ready_For_Transfer : Bool;
         Ready_For_Transfer_Ena : Bool;
         Tank_Available : Bool;
         Transfer_On_Prog : Bool;
      END_STRUCT;
      alwaysON : Bool;
      L_Hys_Abs : Real;
      Hys_Level_HL : Real;
      Hys_Level_ML : Real;
      Hys_Level_LL : Real;
      r : Struct
         PosE1 : Bool;
         PosE2 : Bool;
         PosE3 : Bool;
         PosE4 : Bool;
         PosE5 : Bool;
         PosE6 : Bool;
         PosE7 : Bool;
         PosE8 : Bool;
         PosE9 : Bool;
         PosE10 : Bool;
         PosE11 : Bool;
         PosE12 : Bool;
         PosE13 : Bool;
         PosE14 : Bool;
         PosE15 : Bool;
         PosE16 : Bool;
         PosE17 : Bool;
         PosE18 : Bool;
         PosE19 : Bool;
         PosE20 : Bool;
         PosE21 : Bool;
         PosE22 : Bool;
         PosE23 : Bool;
         PosE24 : Bool;
         PosE25 : Bool;
         PosE26 : Bool;
         PosE27 : Bool;
         PosE28 : Bool;
         PosE29 : Bool;
         PosE30 : Bool;
         PosE31 : Bool;
         PosE32 : Bool;
      END_STRUCT;
      Actuator : Struct
         AV_Inload : Bool;
         AV_Outlet : Bool;
         AV_Transfer : Bool;
         AV_CIP_Tank : Bool;
         AV_CIP_Line : Bool;
         P_Transfer : Bool;
         P_Inload : Bool;
         P_CIP : Bool;
         LCS_OnOff : Bool;
      END_STRUCT;
      FlushingTim : TON_TIME;
      SPumpTim { S7_SetPoint := 'True'} : TON_TIME;
      AVinloadTim { S7_SetPoint := 'True'} : TON_TIME;
      Pump_TF_On_Time { S7_SetPoint := 'True'} : TON_TIME;
   END_VAR
   VAR_TEMP   // added for the SCL form of the ladder/FBD networks
      _w1 : Bool;
      _w2 : Bool;
   END_VAR
BEGIN

REGION Network 1: Always_ON
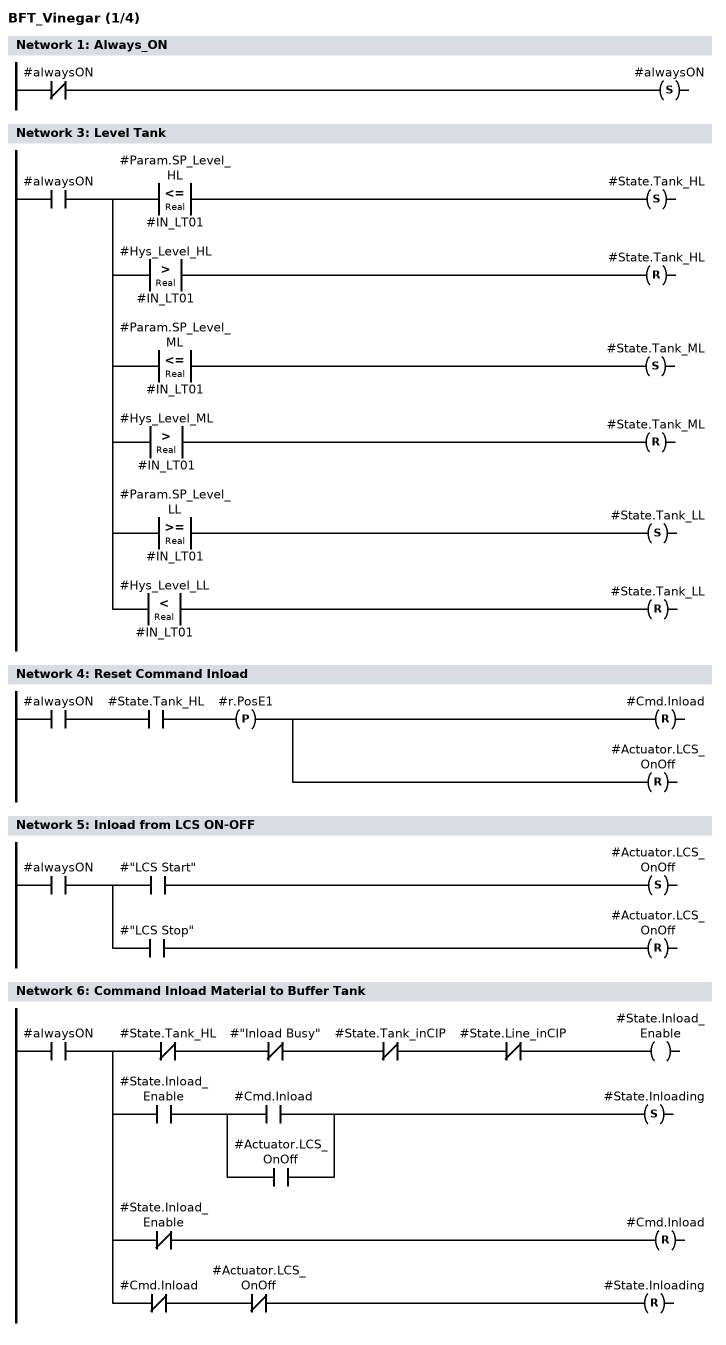
   RUNG wire#powerrail
      I_Contact( #alwaysON )
      S_Coil( #alwaysON )
   END_RUNG
   // the same network as SCL:
   IF NOT #alwaysON THEN #alwaysON := TRUE; END_IF;
END_REGION

NETWORK
TITLE = Hys Calculation
//Level Hys Absolute
      L     #Param.L_Hi_Lim;
      L     #Param.L_Lo_Lim;
      -R;
      L     100.0;
      /R;
      L     #Param.L_Hys;
      *R;
      T     #L_Hys_Abs;
//Tank High Level
      L     #Param.SP_Level_HL;
      L     #L_Hys_Abs;
      -R;
      T     #Hys_Level_HL;
//Tank Mid Level
      L     #Param.SP_Level_ML;
      L     #L_Hys_Abs;
      -R;
      T     #Hys_Level_ML;
//Tank Low Level
      L     #Param.SP_Level_LL;
      L     #L_Hys_Abs;
      +R;
      T     #Hys_Level_LL;


REGION Network 3: Level Tank
   RUNG wire#powerrail
      Contact( #alwaysON )
      wire#w1
      { S7_Templates := "SrcType := Real" } LE_Contact(in1 := #Param.SP_Level_HL, in2 := #IN_LT01)
      S_Coil( #State.Tank_HL )
   END_RUNG
   RUNG wire#w1
      { S7_Templates := "SrcType := Real" } GT_Contact(in1 := #Hys_Level_HL, in2 := #IN_LT01)
      R_Coil( #State.Tank_HL )
   END_RUNG
   RUNG wire#w1
      { S7_Templates := "SrcType := Real" } LE_Contact(in1 := #Param.SP_Level_ML, in2 := #IN_LT01)
      S_Coil( #State.Tank_ML )
   END_RUNG
   RUNG wire#w1
      { S7_Templates := "SrcType := Real" } GT_Contact(in1 := #Hys_Level_ML, in2 := #IN_LT01)
      R_Coil( #State.Tank_ML )
   END_RUNG
   RUNG wire#w1
      { S7_Templates := "SrcType := Real" } GE_Contact(in1 := #Param.SP_Level_LL, in2 := #IN_LT01)
      S_Coil( #State.Tank_LL )
   END_RUNG
   RUNG wire#w1
      { S7_Templates := "SrcType := Real" } LT_Contact(in1 := #Hys_Level_LL, in2 := #IN_LT01)
      R_Coil( #State.Tank_LL )
   END_RUNG
   // the same network as SCL:
   IF #alwaysON AND (#Param.SP_Level_HL <= #IN_LT01) THEN #State.Tank_HL := TRUE; END_IF;
   IF #alwaysON AND (#Hys_Level_HL > #IN_LT01) THEN #State.Tank_HL := FALSE; END_IF;
   IF #alwaysON AND (#Param.SP_Level_ML <= #IN_LT01) THEN #State.Tank_ML := TRUE; END_IF;
   IF #alwaysON AND (#Hys_Level_ML > #IN_LT01) THEN #State.Tank_ML := FALSE; END_IF;
   IF #alwaysON AND (#Param.SP_Level_LL >= #IN_LT01) THEN #State.Tank_LL := TRUE; END_IF;
   IF #alwaysON AND (#Hys_Level_LL < #IN_LT01) THEN #State.Tank_LL := FALSE; END_IF;
END_REGION

REGION Network 4: Reset Command Inload
   RUNG wire#powerrail
      Contact( #alwaysON )
      Contact( #State.Tank_HL )
      P_Trig( #r.PosE1 )
      wire#w1
      R_Coil( #Cmd.Inload )
   END_RUNG
   RUNG wire#w1
      R_Coil( #Actuator.LCS_OnOff )
   END_RUNG
   // the same network as SCL:
   #_w1 := #alwaysON AND #State.Tank_HL;
   #_w2 := #_w1 AND NOT #r.PosE1;   // rising edge
   #r.PosE1 := #_w1;
   IF #_w2 THEN
       #Cmd.Inload := FALSE;
       #Actuator.LCS_OnOff := FALSE;
   END_IF;
END_REGION

REGION Network 5: Inload from LCS ON-OFF
   RUNG wire#powerrail
      Contact( #alwaysON )
      wire#w1
      Contact( #"LCS Start" )
      S_Coil( #Actuator.LCS_OnOff )
   END_RUNG
   RUNG wire#w1
      Contact( #"LCS Stop" )
      R_Coil( #Actuator.LCS_OnOff )
   END_RUNG
   // the same network as SCL:
   IF #alwaysON AND #"LCS Start" THEN #Actuator.LCS_OnOff := TRUE; END_IF;
   IF #alwaysON AND #"LCS Stop" THEN #Actuator.LCS_OnOff := FALSE; END_IF;
END_REGION

REGION Network 6: Command Inload Material to Buffer Tank
   RUNG wire#powerrail
      Contact( #alwaysON )
      wire#w1
      I_Contact( #State.Tank_HL )
      I_Contact( #"Inload Busy" )
      I_Contact( #State.Tank_inCIP )
      I_Contact( #State.Line_inCIP )
      Coil( #State.Inload_Enable )
   END_RUNG
   RUNG wire#w1
      Contact( #State.Inload_Enable )
      wire#w2
      Contact( #Cmd.Inload )
      wire#w3
      S_Coil( #State.Inloading )
   END_RUNG
   RUNG wire#w2
      Contact( #Actuator.LCS_OnOff )
   END_RUNG wire#w3
   RUNG wire#w1
      I_Contact( #State.Inload_Enable )
      R_Coil( #Cmd.Inload )
   END_RUNG
   RUNG wire#w1
      I_Contact( #Cmd.Inload )
      I_Contact( #Actuator.LCS_OnOff )
      R_Coil( #State.Inloading )
   END_RUNG
   // the same network as SCL:
   #State.Inload_Enable := #alwaysON AND NOT #State.Tank_HL AND NOT #"Inload Busy" AND NOT #State.Tank_inCIP AND NOT #State.Line_inCIP;
   IF #alwaysON AND #State.Inload_Enable AND (#Cmd.Inload OR #Actuator.LCS_OnOff) THEN
       #State.Inloading := TRUE;
   END_IF;
   IF #alwaysON AND NOT #State.Inload_Enable THEN #Cmd.Inload := FALSE; END_IF;
   IF #alwaysON AND NOT #Cmd.Inload AND NOT #Actuator.LCS_OnOff THEN #State.Inloading := FALSE; END_IF;
END_REGION

REGION Network 7: Tank Ready for Transfer to Blending
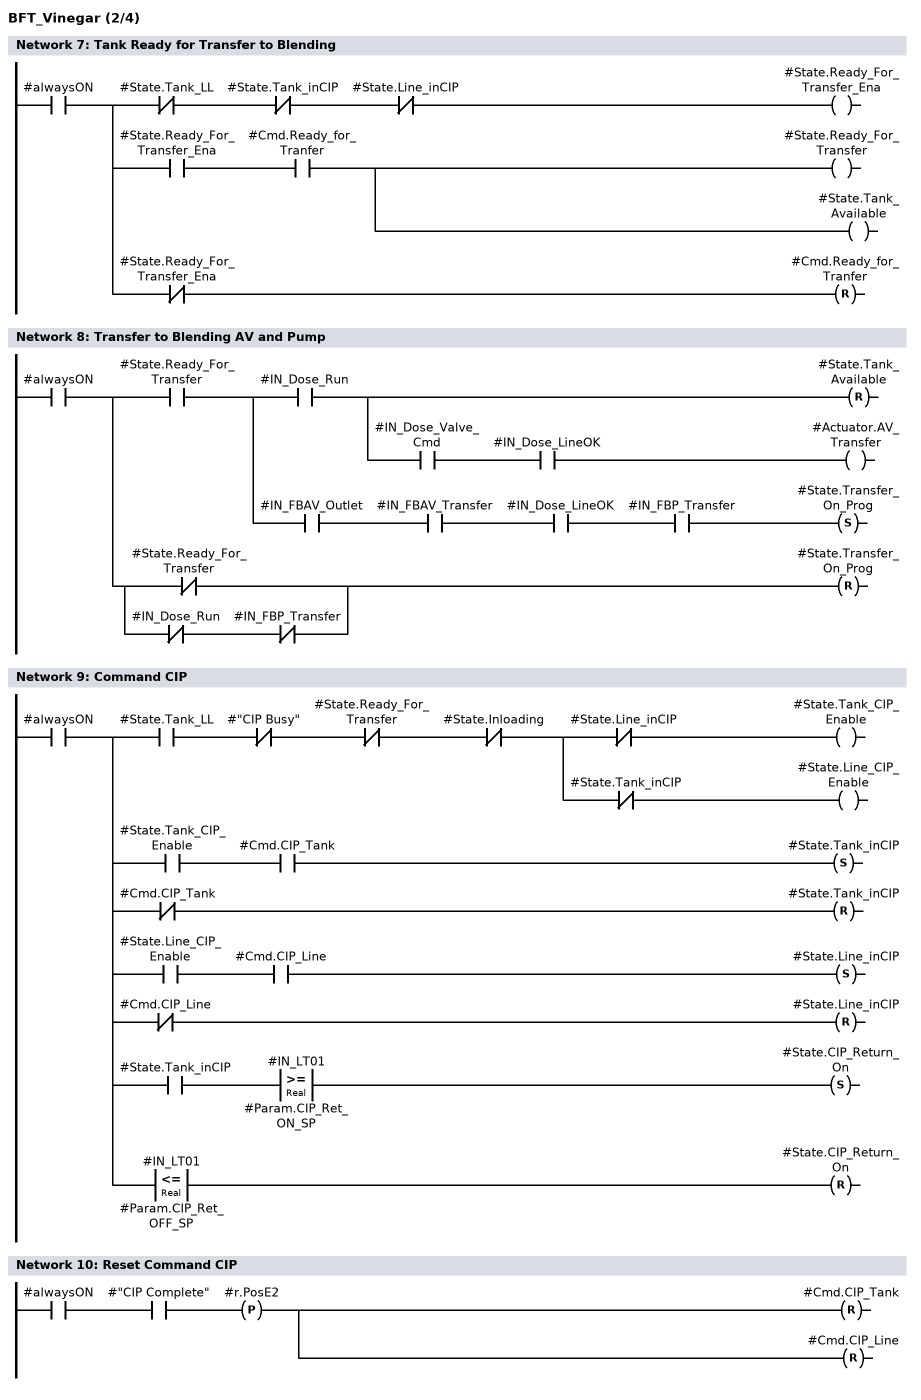
   RUNG wire#powerrail
      Contact( #alwaysON )
      wire#w1
      I_Contact( #State.Tank_LL )
      I_Contact( #State.Tank_inCIP )
      I_Contact( #State.Line_inCIP )
      Coil( #State.Ready_For_Transfer_Ena )
   END_RUNG
   RUNG wire#w1
      Contact( #State.Ready_For_Transfer_Ena )
      Contact( #Cmd.Ready_for_Tranfer )
      wire#w2
      Coil( #State.Ready_For_Transfer )
   END_RUNG
   RUNG wire#w2
      Coil( #State.Tank_Available )
   END_RUNG
   RUNG wire#w1
      I_Contact( #State.Ready_For_Transfer_Ena )
      R_Coil( #Cmd.Ready_for_Tranfer )
   END_RUNG
   // the same network as SCL:
   #State.Ready_For_Transfer_Ena := #alwaysON AND NOT #State.Tank_LL AND NOT #State.Tank_inCIP AND NOT #State.Line_inCIP;
   #State.Ready_For_Transfer := #alwaysON AND #State.Ready_For_Transfer_Ena AND #Cmd.Ready_for_Tranfer;
   #State.Tank_Available := #State.Ready_For_Transfer;
   IF #alwaysON AND NOT #State.Ready_For_Transfer_Ena THEN #Cmd.Ready_for_Tranfer := FALSE; END_IF;
END_REGION

REGION Network 8: Transfer to Blending AV and Pump
   RUNG wire#powerrail
      Contact( #alwaysON )
      wire#w1
      Contact( #State.Ready_For_Transfer )
      wire#w2
      Contact( #IN_Dose_Run )
      wire#w3
      R_Coil( #State.Tank_Available )
   END_RUNG
   RUNG wire#w3
      Contact( #IN_Dose_Valve_Cmd )
      Contact( #IN_Dose_LineOK )
      Coil( #Actuator.AV_Transfer )
   END_RUNG
   RUNG wire#w2
      Contact( #IN_FBAV_Outlet )
      Contact( #IN_FBAV_Transfer )
      Contact( #IN_Dose_LineOK )
      Contact( #IN_FBP_Transfer )
      S_Coil( #State.Transfer_On_Prog )
   END_RUNG
   RUNG wire#w1
      I_Contact( #State.Ready_For_Transfer )
      wire#w4
      R_Coil( #State.Transfer_On_Prog )
   END_RUNG
   RUNG wire#w1
      I_Contact( #IN_Dose_Run )
      I_Contact( #IN_FBP_Transfer )
   END_RUNG wire#w4
   // the same network as SCL:
   #_w1 := #alwaysON AND #State.Ready_For_Transfer;
   #_w2 := #_w1 AND #IN_Dose_Run;
   IF #_w2 THEN #State.Tank_Available := FALSE; END_IF;
   #Actuator.AV_Transfer := #_w2 AND #IN_Dose_Valve_Cmd AND #IN_Dose_LineOK;
   IF #_w1 AND #IN_FBAV_Outlet AND #IN_FBAV_Transfer AND #IN_Dose_LineOK AND #IN_FBP_Transfer THEN
       #State.Transfer_On_Prog := TRUE;
   END_IF;
   IF #alwaysON AND (NOT #State.Ready_For_Transfer OR (NOT #IN_Dose_Run AND NOT #IN_FBP_Transfer)) THEN
       #State.Transfer_On_Prog := FALSE;
   END_IF;
END_REGION

REGION Network 9: Command CIP
   RUNG wire#powerrail
      Contact( #alwaysON )
      wire#w1
      Contact( #State.Tank_LL )
      I_Contact( #"CIP Busy" )
      I_Contact( #State.Ready_For_Transfer )
      I_Contact( #State.Inloading )
      wire#w2
      I_Contact( #State.Line_inCIP )
      Coil( #State.Tank_CIP_Enable )
   END_RUNG
   RUNG wire#w2
      I_Contact( #State.Tank_inCIP )
      Coil( #State.Line_CIP_Enable )
   END_RUNG
   RUNG wire#w1
      Contact( #State.Tank_CIP_Enable )
      Contact( #Cmd.CIP_Tank )
      S_Coil( #State.Tank_inCIP )
   END_RUNG
   RUNG wire#w1
      I_Contact( #Cmd.CIP_Tank )
      R_Coil( #State.Tank_inCIP )
   END_RUNG
   RUNG wire#w1
      Contact( #State.Line_CIP_Enable )
      Contact( #Cmd.CIP_Line )
      S_Coil( #State.Line_inCIP )
   END_RUNG
   RUNG wire#w1
      I_Contact( #Cmd.CIP_Line )
      R_Coil( #State.Line_inCIP )
   END_RUNG
   RUNG wire#w1
      Contact( #State.Tank_inCIP )
      { S7_Templates := "SrcType := Real" } GE_Contact(in1 := #IN_LT01, in2 := #Param.CIP_Ret_ON_SP)
      S_Coil( #State.CIP_Return_On )
   END_RUNG
   RUNG wire#w1
      { S7_Templates := "SrcType := Real" } LE_Contact(in1 := #IN_LT01, in2 := #Param.CIP_Ret_OFF_SP)
      R_Coil( #State.CIP_Return_On )
   END_RUNG
   // the same network as SCL:
   #_w1 := #alwaysON AND #State.Tank_LL AND NOT #"CIP Busy" AND NOT #State.Ready_For_Transfer AND NOT #State.Inloading;
   #State.Tank_CIP_Enable := #_w1 AND NOT #State.Line_inCIP;
   #State.Line_CIP_Enable := #_w1 AND NOT #State.Tank_inCIP;
   IF #alwaysON AND #State.Tank_CIP_Enable AND #Cmd.CIP_Tank THEN #State.Tank_inCIP := TRUE; END_IF;
   IF #alwaysON AND NOT #Cmd.CIP_Tank THEN #State.Tank_inCIP := FALSE; END_IF;
   IF #alwaysON AND #State.Line_CIP_Enable AND #Cmd.CIP_Line THEN #State.Line_inCIP := TRUE; END_IF;
   IF #alwaysON AND NOT #Cmd.CIP_Line THEN #State.Line_inCIP := FALSE; END_IF;
   IF #alwaysON AND #State.Tank_inCIP AND (#IN_LT01 >= #Param.CIP_Ret_ON_SP) THEN
       #State.CIP_Return_On := TRUE;
   END_IF;
   IF #alwaysON AND (#IN_LT01 <= #Param.CIP_Ret_OFF_SP) THEN #State.CIP_Return_On := FALSE; END_IF;
END_REGION

REGION Network 10: Reset Command CIP
   RUNG wire#powerrail
      Contact( #alwaysON )
      Contact( #"CIP Complete" )
      P_Trig( #r.PosE2 )
      wire#w1
      R_Coil( #Cmd.CIP_Tank )
   END_RUNG
   RUNG wire#w1
      R_Coil( #Cmd.CIP_Line )
   END_RUNG
   // the same network as SCL:
   #_w1 := #alwaysON AND #"CIP Complete";
   #_w2 := #_w1 AND NOT #r.PosE2;   // rising edge
   #r.PosE2 := #_w1;
   IF #_w2 THEN
       #Cmd.CIP_Tank := FALSE;
       #Cmd.CIP_Line := FALSE;
   END_IF;
END_REGION

REGION Network 11: CIP Request and CIP Line Open
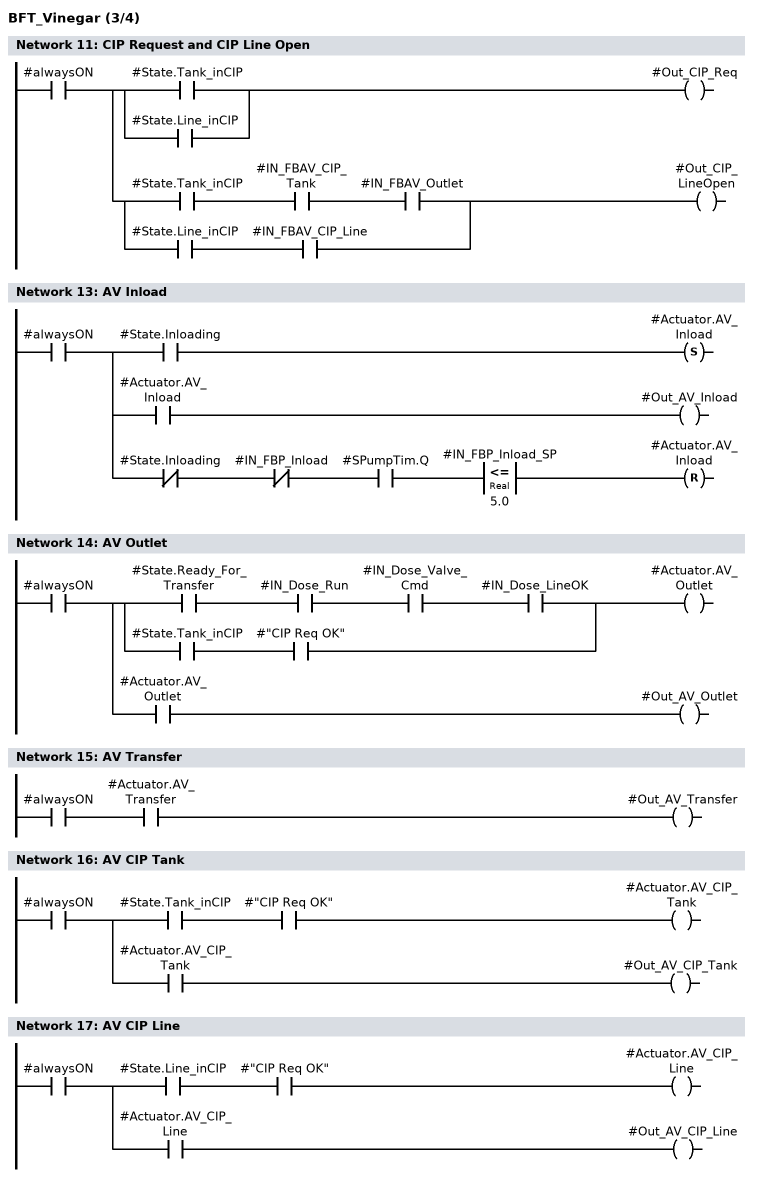
   RUNG wire#powerrail
      Contact( #alwaysON )
      wire#w1
      Contact( #State.Tank_inCIP )
      wire#w2
      Coil( #Out_CIP_Req )
   END_RUNG
   RUNG wire#w1
      Contact( #State.Line_inCIP )
   END_RUNG wire#w2
   RUNG wire#w1
      Contact( #State.Tank_inCIP )
      Contact( #IN_FBAV_CIP_Tank )
      Contact( #IN_FBAV_Outlet )
      wire#w3
      Coil( #Out_CIP_LineOpen )
   END_RUNG
   RUNG wire#w1
      Contact( #State.Line_inCIP )
      Contact( #IN_FBAV_CIP_Line )
   END_RUNG wire#w3
   // the same network as SCL:
   #Out_CIP_Req := #alwaysON AND (#State.Tank_inCIP OR #State.Line_inCIP);
   #Out_CIP_LineOpen := #alwaysON AND ((#State.Tank_inCIP AND #IN_FBAV_CIP_Tank AND #IN_FBAV_Outlet) OR (#State.Line_inCIP AND #IN_FBAV_CIP_Line));
END_REGION

REGION Network 13: AV Inload
   RUNG wire#powerrail
      Contact( #alwaysON )
      wire#w1
      Contact( #State.Inloading )
      S_Coil( #Actuator.AV_Inload )
   END_RUNG
   RUNG wire#w1
      Contact( #Actuator.AV_Inload )
      Coil( #Out_AV_Inload )
   END_RUNG
   RUNG wire#w1
      I_Contact( #State.Inloading )
      I_Contact( #IN_FBP_Inload )
      Contact( #SPumpTim.Q )
      { S7_Templates := "SrcType := Real" } LE_Contact(in1 := #IN_FBP_Inload_SP, in2 := 5.0)
      R_Coil( #Actuator.AV_Inload )
   END_RUNG
   // the same network as SCL:
   IF #alwaysON AND #State.Inloading THEN #Actuator.AV_Inload := TRUE; END_IF;
   #Out_AV_Inload := #alwaysON AND #Actuator.AV_Inload;
   IF #alwaysON AND NOT #State.Inloading AND NOT #IN_FBP_Inload AND #SPumpTim.Q AND (#IN_FBP_Inload_SP <= 5.0) THEN
       #Actuator.AV_Inload := FALSE;
   END_IF;
END_REGION

REGION Network 14: AV Outlet
   RUNG wire#powerrail
      Contact( #alwaysON )
      wire#w1
      Contact( #State.Ready_For_Transfer )
      Contact( #IN_Dose_Run )
      Contact( #IN_Dose_Valve_Cmd )
      Contact( #IN_Dose_LineOK )
      wire#w2
      Coil( #Actuator.AV_Outlet )
   END_RUNG
   RUNG wire#w1
      Contact( #State.Tank_inCIP )
      Contact( #"CIP Req OK" )
   END_RUNG wire#w2
   RUNG wire#w1
      Contact( #Actuator.AV_Outlet )
      Coil( #Out_AV_Outlet )
   END_RUNG
   // the same network as SCL:
   #Actuator.AV_Outlet := #alwaysON AND ((#State.Ready_For_Transfer AND #IN_Dose_Run AND #IN_Dose_Valve_Cmd AND #IN_Dose_LineOK) OR (#State.Tank_inCIP AND #"CIP Req OK"));
   #Out_AV_Outlet := #alwaysON AND #Actuator.AV_Outlet;
END_REGION

REGION Network 15: AV Transfer
   RUNG wire#powerrail
      Contact( #alwaysON )
      Contact( #Actuator.AV_Transfer )
      Coil( #Out_AV_Transfer )
   END_RUNG
   // the same network as SCL:
   #Out_AV_Transfer := #alwaysON AND #Actuator.AV_Transfer;
END_REGION

REGION Network 16: AV CIP Tank
   RUNG wire#powerrail
      Contact( #alwaysON )
      wire#w1
      Contact( #State.Tank_inCIP )
      Contact( #"CIP Req OK" )
      Coil( #Actuator.AV_CIP_Tank )
   END_RUNG
   RUNG wire#w1
      Contact( #Actuator.AV_CIP_Tank )
      Coil( #Out_AV_CIP_Tank )
   END_RUNG
   // the same network as SCL:
   #Actuator.AV_CIP_Tank := #alwaysON AND #State.Tank_inCIP AND #"CIP Req OK";
   #Out_AV_CIP_Tank := #alwaysON AND #Actuator.AV_CIP_Tank;
END_REGION

REGION Network 17: AV CIP Line
   RUNG wire#powerrail
      Contact( #alwaysON )
      wire#w1
      Contact( #State.Line_inCIP )
      Contact( #"CIP Req OK" )
      Coil( #Actuator.AV_CIP_Line )
   END_RUNG
   RUNG wire#w1
      Contact( #Actuator.AV_CIP_Line )
      Coil( #Out_AV_CIP_Line )
   END_RUNG
   // the same network as SCL:
   #Actuator.AV_CIP_Line := #alwaysON AND #State.Line_inCIP AND #"CIP Req OK";
   #Out_AV_CIP_Line := #alwaysON AND #Actuator.AV_CIP_Line;
END_REGION

REGION Network 19: Pump Inload
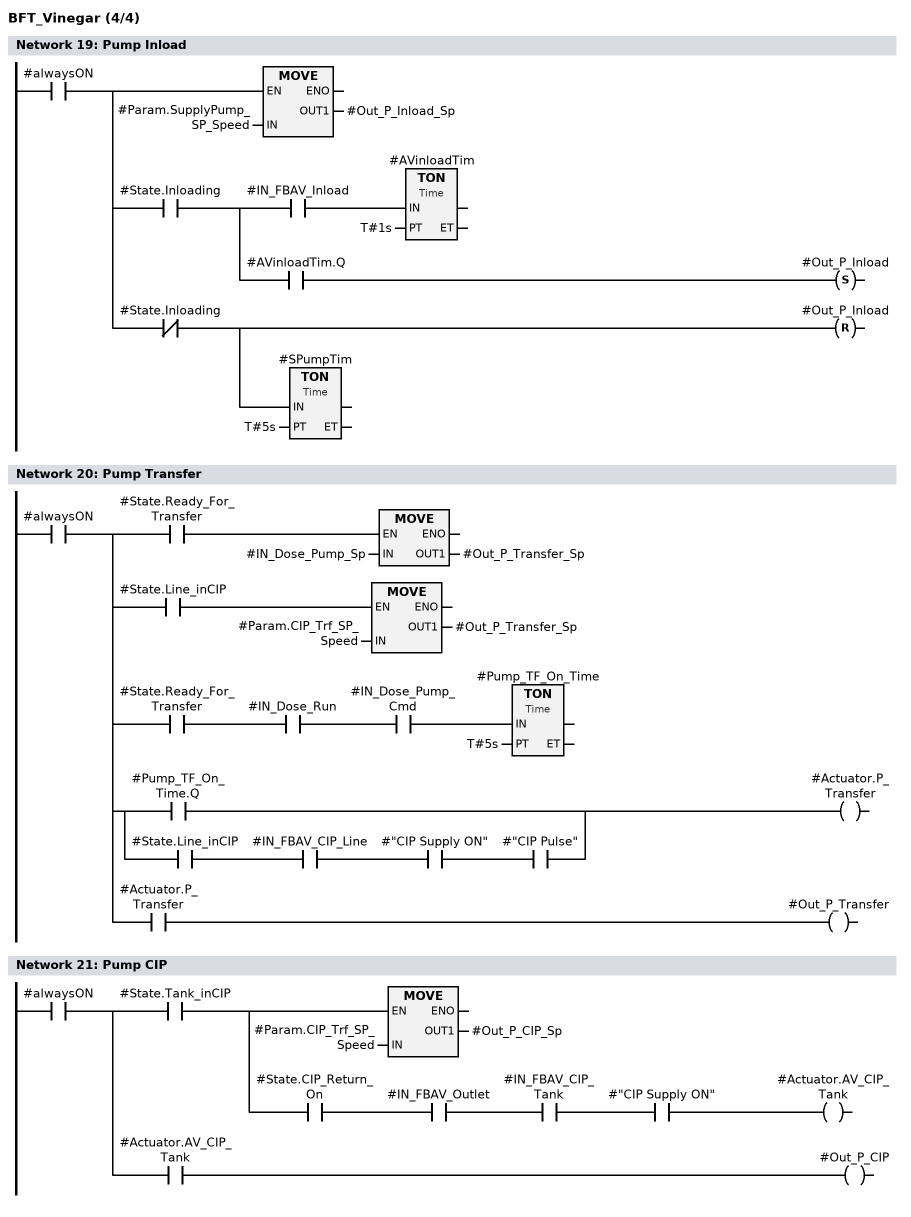
   RUNG wire#powerrail
      Contact( #alwaysON )
      wire#w1
      Move(in := #Param.SupplyPump_SP_Speed, out1 => #Out_P_Inload_Sp)
   END_RUNG
   RUNG wire#w1
      Contact( #State.Inloading )
      wire#w2
      Contact( #IN_FBAV_Inload )
      { S7_Templates := "time_type := Time" } #AVinloadTim.TON(pt := T#1s, et =>)
   END_RUNG
   RUNG wire#w2
      Contact( #AVinloadTim.Q )
      S_Coil( #Out_P_Inload )
   END_RUNG
   RUNG wire#w1
      I_Contact( #State.Inloading )
      wire#w3
      R_Coil( #Out_P_Inload )
   END_RUNG
   RUNG wire#w3
      { S7_Templates := "time_type := Time" } #SPumpTim.TON(pt := T#5s, et =>)
   END_RUNG
   // the same network as SCL:
   IF #alwaysON THEN #Out_P_Inload_Sp := #Param.SupplyPump_SP_Speed; END_IF;
   #_w1 := #alwaysON AND #State.Inloading;
   #AVinloadTim(IN := #_w1 AND #IN_FBAV_Inload, PT := T#1s);   // TON
   IF #_w1 AND #AVinloadTim.Q THEN #Out_P_Inload := TRUE; END_IF;
   #_w2 := #alwaysON AND NOT #State.Inloading;
   IF #_w2 THEN #Out_P_Inload := FALSE; END_IF;
   #SPumpTim(IN := #_w2, PT := T#5s);   // TON
END_REGION

REGION Network 20: Pump Transfer
   RUNG wire#powerrail
      Contact( #alwaysON )
      wire#w1
      Contact( #State.Ready_For_Transfer )
      Move(in := #IN_Dose_Pump_Sp, out1 => #Out_P_Transfer_Sp)
   END_RUNG
   RUNG wire#w1
      Contact( #State.Line_inCIP )
      Move(in := #Param.CIP_Trf_SP_Speed, out1 => #Out_P_Transfer_Sp)
   END_RUNG
   RUNG wire#w1
      Contact( #State.Ready_For_Transfer )
      Contact( #IN_Dose_Run )
      Contact( #IN_Dose_Pump_Cmd )
      { S7_Templates := "time_type := Time" } #Pump_TF_On_Time.TON(pt := T#5s, et =>)
   END_RUNG
   RUNG wire#w1
      Contact( #Pump_TF_On_Time.Q )
      wire#w2
      Coil( #Actuator.P_Transfer )
   END_RUNG
   RUNG wire#w1
      Contact( #State.Line_inCIP )
      Contact( #IN_FBAV_CIP_Line )
      Contact( #"CIP Supply ON" )
      Contact( #"CIP Pulse" )
   END_RUNG wire#w2
   RUNG wire#w1
      Contact( #Actuator.P_Transfer )
      Coil( #Out_P_Transfer )
   END_RUNG
   // the same network as SCL:
   IF #alwaysON AND #State.Ready_For_Transfer THEN #Out_P_Transfer_Sp := #IN_Dose_Pump_Sp; END_IF;
   IF #alwaysON AND #State.Line_inCIP THEN #Out_P_Transfer_Sp := #Param.CIP_Trf_SP_Speed; END_IF;
   #Pump_TF_On_Time(IN := #alwaysON AND #State.Ready_For_Transfer AND #IN_Dose_Run AND #IN_Dose_Pump_Cmd,   // TON
                    PT := T#5s);
   #Actuator.P_Transfer := #alwaysON AND (#Pump_TF_On_Time.Q OR (#State.Line_inCIP AND #IN_FBAV_CIP_Line AND #"CIP Supply ON" AND #"CIP Pulse"));
   #Out_P_Transfer := #alwaysON AND #Actuator.P_Transfer;
END_REGION

REGION Network 21: Pump CIP
   RUNG wire#powerrail
      Contact( #alwaysON )
      wire#w1
      Contact( #State.Tank_inCIP )
      wire#w2
      Move(in := #Param.CIP_Trf_SP_Speed, out1 => #Out_P_CIP_Sp)
   END_RUNG
   RUNG wire#w2
      Contact( #State.CIP_Return_On )
      Contact( #IN_FBAV_Outlet )
      Contact( #IN_FBAV_CIP_Tank )
      Contact( #"CIP Supply ON" )
      Coil( #Actuator.AV_CIP_Tank )
   END_RUNG
   RUNG wire#w1
      Contact( #Actuator.AV_CIP_Tank )
      Coil( #Out_P_CIP )
   END_RUNG
   // the same network as SCL:
   #_w1 := #alwaysON AND #State.Tank_inCIP;
   IF #_w1 THEN #Out_P_CIP_Sp := #Param.CIP_Trf_SP_Speed; END_IF;
   #Actuator.AV_CIP_Tank := #_w1 AND #State.CIP_Return_On AND #IN_FBAV_Outlet AND #IN_FBAV_CIP_Tank AND #"CIP Supply ON";
   #Out_P_CIP := #alwaysON AND #Actuator.AV_CIP_Tank;
END_REGION
END_FUNCTION_BLOCK

FUNCTION_BLOCK "Hot_Water"   // FB366, LAD
{ S7_Optimized_Access := 'TRUE' }
VERSION : 0.1
// stored: AutoNumber false, IsIECCheckEnabled false, IsRetainMemResEnabled false, MemoryReserve 100, SetENOAutomatically false, UDAEnableTagReadback false
   VAR_INPUT
      IN_FBAV_Inload : Bool;
      IN_FBAV_Outlet : Bool;
      IN_FBAV_Transfer : Bool;
      IN_FBP_Transfer : Bool;
      IN_FBP_Transfer_SP : Real;
      IN_Dose_Run : Bool;
      IN_Dose_Held : Bool;
      IN_Dose_Complete : Bool;
      IN_Dose_Header_1 : Bool;
      IN_Dose_Header_2 : Bool;
      IN_Dose_Valve_Cmd : Bool;
      IN_Dose_Pump_Cmd : Bool;
      IN_Dose_Pump_Sp : Real;
      IN_Dose_LineOK : Bool;
      IN_Low_Level : Bool;
      IN_Med_Level : Bool;
      IN_High_Level : Bool;
      IN_FBCV : Bool;
      "IN_FBCV_Act%" : Real;
      IN_Temperature : Real;
   END_VAR
   VAR_OUTPUT
      Out_AV_Inload : Bool;
      Out_AV_Outlet : Bool;
      Out_AV_Transfer : Bool;
      Out_P_Transfer : Bool;
      Out_P_Transfer_Sp : Real;
      OUT_CV : Bool;
      Out_Temp_Act : Real;
      Out_Temp_Sp : Real;
   END_VAR
   VAR
      Cmd : Struct
         Inload_Start : Bool;
         Inload_Mode : Bool := 1;   // 0 : Manual ;; 1 : Auto
         ReadyForTransfer : Bool;
         Transfer_Mode : Bool;   // 0 : By Timer ;; 1 : By Quantity
      END_STRUCT;
   END_VAR
   VAR RETAIN
      Param : Struct
         Temperature_SP : Real := 50.0;
      END_STRUCT;
   END_VAR
   VAR
      State : Struct
         Tank_LL : Bool;
         Tank_ML : Bool;
         Tank_HL : Bool;
         Inload_EN : Bool;
         Inload_Aut : Bool;
         Inloading : Bool;
         Ready_For_Transfer_EN : Bool;
         Ready_For_Transfer : Bool;
         Tank_Available : Bool;
         Transfer_on_Prog : Bool;
      END_STRUCT;
      alwaysON : Bool;
      r : Struct
         PosE1 : Bool;
         PosE2 : Bool;
         PosE3 : Bool;
         PosE4 : Bool;
         PosE5 : Bool;
         PosE6 : Bool;
         PosE7 : Bool;
         PosE8 : Bool;
         PosE9 : Bool;
         PosE10 : Bool;
         PosE11 : Bool;
         PosE12 : Bool;
         PosE13 : Bool;
         PosE14 : Bool;
         PosE15 : Bool;
         PosE16 : Bool;
         PosE17 : Bool;
         PosE18 : Bool;
         PosE19 : Bool;
         PosE20 : Bool;
         PosE21 : Bool;
         PosE22 : Bool;
         PosE23 : Bool;
         PosE24 : Bool;
         PosE25 : Bool;
         PosE26 : Bool;
         PosE27 : Bool;
         PosE28 : Bool;
         PosE29 : Bool;
         PosE30 : Bool;
         PosE31 : Bool;
         PosE32 : Bool;
      END_STRUCT;
      Actuator : Struct
         AV_Inload : Bool;
         AV_Outlet : Bool;
         AV_Transfer : Bool;
         AV_CIP_Tank : Bool;
         AV_CIP_Line : Bool;
         P_Transfer : Bool;
         P_Inload : Bool;
         P_CIP : Bool;
         CV : Bool;
      END_STRUCT;
      SPumpTim { S7_SetPoint := 'True'} : TON_TIME;
   END_VAR
   VAR_TEMP   // added for the SCL form of the ladder/FBD networks
      _w1 : Bool;
      _w2 : Bool;
   END_VAR
BEGIN

REGION Network 1: Always_ON
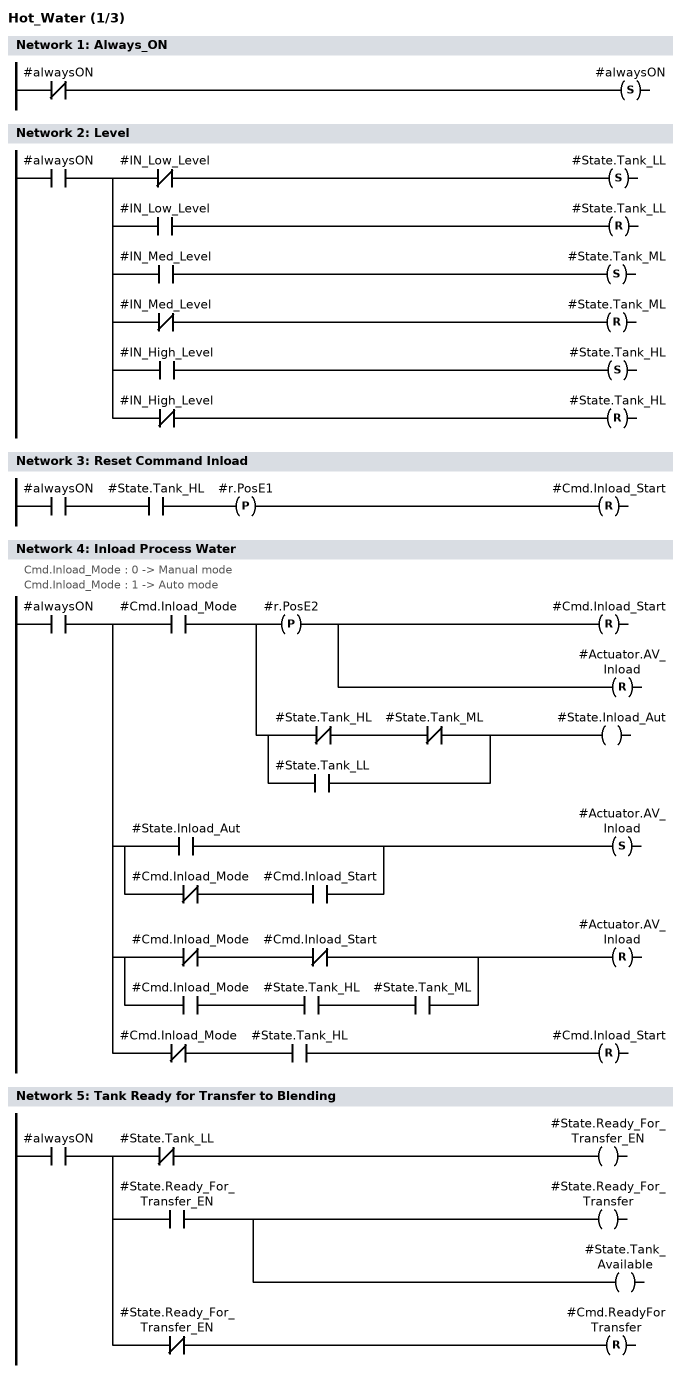
   RUNG wire#powerrail
      I_Contact( #alwaysON )
      S_Coil( #alwaysON )
   END_RUNG
   // the same network as SCL:
   IF NOT #alwaysON THEN #alwaysON := TRUE; END_IF;
END_REGION

REGION Network 2: Level
   RUNG wire#powerrail
      Contact( #alwaysON )
      wire#w1
      I_Contact( #IN_Low_Level )
      S_Coil( #State.Tank_LL )
   END_RUNG
   RUNG wire#w1
      Contact( #IN_Low_Level )
      R_Coil( #State.Tank_LL )
   END_RUNG
   RUNG wire#w1
      Contact( #IN_Med_Level )
      S_Coil( #State.Tank_ML )
   END_RUNG
   RUNG wire#w1
      I_Contact( #IN_Med_Level )
      R_Coil( #State.Tank_ML )
   END_RUNG
   RUNG wire#w1
      Contact( #IN_High_Level )
      S_Coil( #State.Tank_HL )
   END_RUNG
   RUNG wire#w1
      I_Contact( #IN_High_Level )
      R_Coil( #State.Tank_HL )
   END_RUNG
   // the same network as SCL:
   IF #alwaysON AND NOT #IN_Low_Level THEN #State.Tank_LL := TRUE; END_IF;
   IF #alwaysON AND #IN_Low_Level THEN #State.Tank_LL := FALSE; END_IF;
   IF #alwaysON AND #IN_Med_Level THEN #State.Tank_ML := TRUE; END_IF;
   IF #alwaysON AND NOT #IN_Med_Level THEN #State.Tank_ML := FALSE; END_IF;
   IF #alwaysON AND #IN_High_Level THEN #State.Tank_HL := TRUE; END_IF;
   IF #alwaysON AND NOT #IN_High_Level THEN #State.Tank_HL := FALSE; END_IF;
END_REGION

REGION Network 3: Reset Command Inload
   RUNG wire#powerrail
      Contact( #alwaysON )
      Contact( #State.Tank_HL )
      P_Trig( #r.PosE1 )
      R_Coil( #Cmd.Inload_Start )
   END_RUNG
   // the same network as SCL:
   #_w1 := #alwaysON AND #State.Tank_HL;
   #_w2 := #_w1 AND NOT #r.PosE1;   // rising edge
   #r.PosE1 := #_w1;
   IF #_w2 THEN #Cmd.Inload_Start := FALSE; END_IF;
END_REGION

REGION Network 4: Inload Process Water
   // Cmd.Inload_Mode : 0 -> Manual mode
   // Cmd.Inload_Mode : 1 -> Auto mode
   RUNG wire#powerrail
      Contact( #alwaysON )
      wire#w1
      Contact( #Cmd.Inload_Mode )
      wire#w2
      P_Trig( #r.PosE2 )
      wire#w3
      R_Coil( #Cmd.Inload_Start )
   END_RUNG
   RUNG wire#w3
      R_Coil( #Actuator.AV_Inload )
   END_RUNG
   RUNG wire#w2
      I_Contact( #State.Tank_HL )
      I_Contact( #State.Tank_ML )
      wire#w4
      Coil( #State.Inload_Aut )
   END_RUNG
   RUNG wire#w2
      Contact( #State.Tank_LL )
   END_RUNG wire#w4
   RUNG wire#w1
      Contact( #State.Inload_Aut )
      wire#w5
      S_Coil( #Actuator.AV_Inload )
   END_RUNG
   RUNG wire#w1
      I_Contact( #Cmd.Inload_Mode )
      Contact( #Cmd.Inload_Start )
   END_RUNG wire#w5
   RUNG wire#w1
      I_Contact( #Cmd.Inload_Mode )
      I_Contact( #Cmd.Inload_Start )
      wire#w6
      R_Coil( #Actuator.AV_Inload )
   END_RUNG
   RUNG wire#w1
      Contact( #Cmd.Inload_Mode )
      Contact( #State.Tank_HL )
      Contact( #State.Tank_ML )
   END_RUNG wire#w6
   RUNG wire#w1
      I_Contact( #Cmd.Inload_Mode )
      Contact( #State.Tank_HL )
      R_Coil( #Cmd.Inload_Start )
   END_RUNG
   // the same network as SCL:
   #_w1 := #alwaysON AND #Cmd.Inload_Mode;
   #_w2 := #_w1 AND NOT #r.PosE2;   // rising edge
   #r.PosE2 := #_w1;
   IF #_w2 THEN
       #Cmd.Inload_Start := FALSE;
       #Actuator.AV_Inload := FALSE;
   END_IF;
   #State.Inload_Aut := #_w1 AND ((NOT #State.Tank_HL AND NOT #State.Tank_ML) OR #State.Tank_LL);
   IF #alwaysON AND (#State.Inload_Aut OR (NOT #Cmd.Inload_Mode AND #Cmd.Inload_Start)) THEN
       #Actuator.AV_Inload := TRUE;
   END_IF;
   IF #alwaysON AND ((NOT #Cmd.Inload_Mode AND NOT #Cmd.Inload_Start) OR (#Cmd.Inload_Mode AND #State.Tank_HL AND #State.Tank_ML)) THEN
       #Actuator.AV_Inload := FALSE;
   END_IF;
   IF #alwaysON AND NOT #Cmd.Inload_Mode AND #State.Tank_HL THEN #Cmd.Inload_Start := FALSE; END_IF;
END_REGION

REGION Network 5: Tank Ready for Transfer to Blending
   RUNG wire#powerrail
      Contact( #alwaysON )
      wire#w1
      I_Contact( #State.Tank_LL )
      Coil( #State.Ready_For_Transfer_EN )
   END_RUNG
   RUNG wire#w1
      Contact( #State.Ready_For_Transfer_EN )
      wire#w2
      Coil( #State.Ready_For_Transfer )
   END_RUNG
   RUNG wire#w2
      Coil( #State.Tank_Available )
   END_RUNG
   RUNG wire#w1
      I_Contact( #State.Ready_For_Transfer_EN )
      R_Coil( #Cmd.ReadyForTransfer )
   END_RUNG
   // the same network as SCL:
   #State.Ready_For_Transfer_EN := #alwaysON AND NOT #State.Tank_LL;
   #State.Ready_For_Transfer := #alwaysON AND #State.Ready_For_Transfer_EN;
   #State.Tank_Available := #State.Ready_For_Transfer;
   IF #alwaysON AND NOT #State.Ready_For_Transfer_EN THEN #Cmd.ReadyForTransfer := FALSE; END_IF;
END_REGION

REGION Network 6: Transfer to Blending AV and Pump
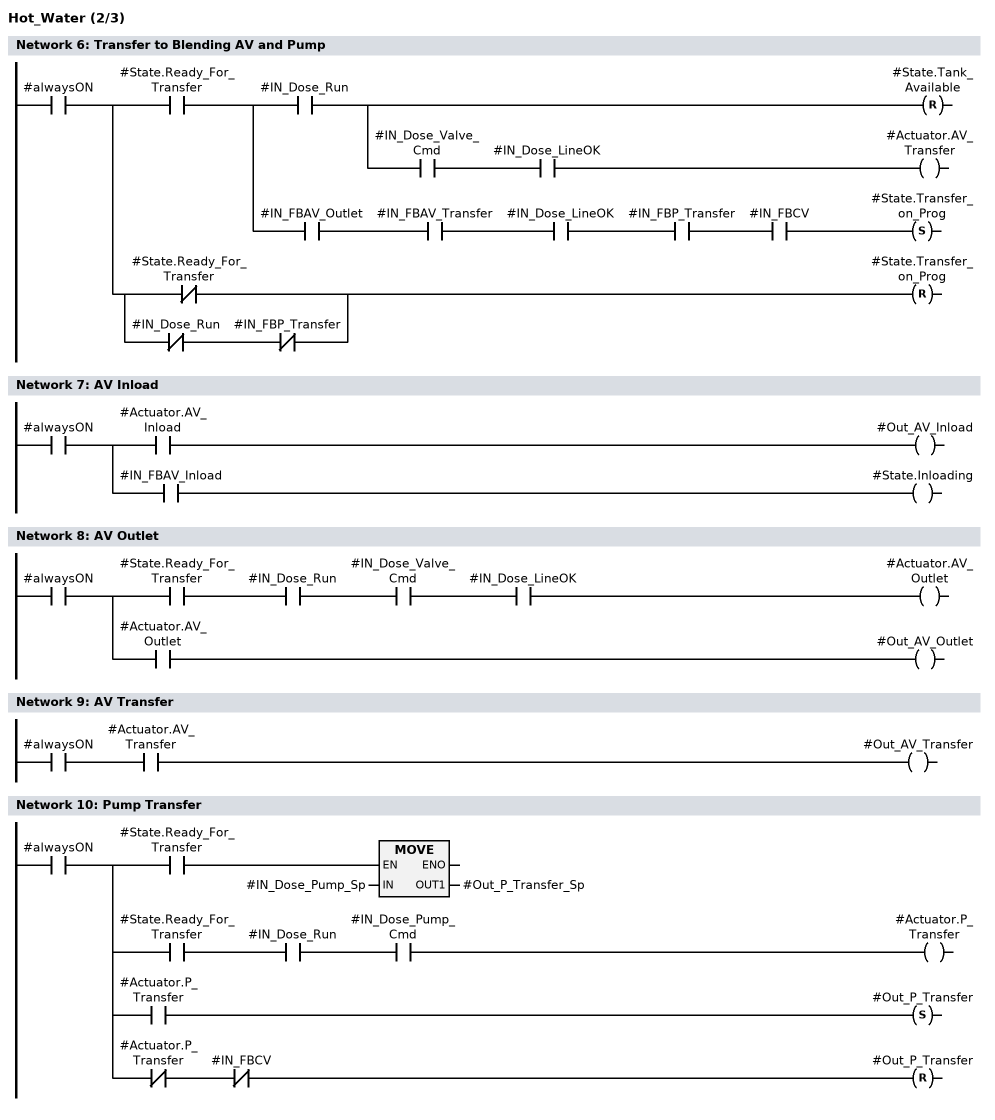
   RUNG wire#powerrail
      Contact( #alwaysON )
      wire#w1
      Contact( #State.Ready_For_Transfer )
      wire#w2
      Contact( #IN_Dose_Run )
      wire#w3
      R_Coil( #State.Tank_Available )
   END_RUNG
   RUNG wire#w3
      Contact( #IN_Dose_Valve_Cmd )
      Contact( #IN_Dose_LineOK )
      Coil( #Actuator.AV_Transfer )
   END_RUNG
   RUNG wire#w2
      Contact( #IN_FBAV_Outlet )
      Contact( #IN_FBAV_Transfer )
      Contact( #IN_Dose_LineOK )
      Contact( #IN_FBP_Transfer )
      Contact( #IN_FBCV )
      S_Coil( #State.Transfer_on_Prog )
   END_RUNG
   RUNG wire#w1
      I_Contact( #State.Ready_For_Transfer )
      wire#w4
      R_Coil( #State.Transfer_on_Prog )
   END_RUNG
   RUNG wire#w1
      I_Contact( #IN_Dose_Run )
      I_Contact( #IN_FBP_Transfer )
   END_RUNG wire#w4
   // the same network as SCL:
   #_w1 := #alwaysON AND #State.Ready_For_Transfer;
   #_w2 := #_w1 AND #IN_Dose_Run;
   IF #_w2 THEN #State.Tank_Available := FALSE; END_IF;
   #Actuator.AV_Transfer := #_w2 AND #IN_Dose_Valve_Cmd AND #IN_Dose_LineOK;
   IF #_w1 AND #IN_FBAV_Outlet AND #IN_FBAV_Transfer AND #IN_Dose_LineOK AND #IN_FBP_Transfer AND #IN_FBCV THEN
       #State.Transfer_on_Prog := TRUE;
   END_IF;
   IF #alwaysON AND (NOT #State.Ready_For_Transfer OR (NOT #IN_Dose_Run AND NOT #IN_FBP_Transfer)) THEN
       #State.Transfer_on_Prog := FALSE;
   END_IF;
END_REGION

REGION Network 7: AV Inload
   RUNG wire#powerrail
      Contact( #alwaysON )
      wire#w1
      Contact( #Actuator.AV_Inload )
      Coil( #Out_AV_Inload )
   END_RUNG
   RUNG wire#w1
      Contact( #IN_FBAV_Inload )
      Coil( #State.Inloading )
   END_RUNG
   // the same network as SCL:
   #Out_AV_Inload := #alwaysON AND #Actuator.AV_Inload;
   #State.Inloading := #alwaysON AND #IN_FBAV_Inload;
END_REGION

REGION Network 8: AV Outlet
   RUNG wire#powerrail
      Contact( #alwaysON )
      wire#w1
      Contact( #State.Ready_For_Transfer )
      Contact( #IN_Dose_Run )
      Contact( #IN_Dose_Valve_Cmd )
      Contact( #IN_Dose_LineOK )
      Coil( #Actuator.AV_Outlet )
   END_RUNG
   RUNG wire#w1
      Contact( #Actuator.AV_Outlet )
      Coil( #Out_AV_Outlet )
   END_RUNG
   // the same network as SCL:
   #Actuator.AV_Outlet := #alwaysON AND #State.Ready_For_Transfer AND #IN_Dose_Run AND #IN_Dose_Valve_Cmd AND #IN_Dose_LineOK;
   #Out_AV_Outlet := #alwaysON AND #Actuator.AV_Outlet;
END_REGION

REGION Network 9: AV Transfer
   RUNG wire#powerrail
      Contact( #alwaysON )
      Contact( #Actuator.AV_Transfer )
      Coil( #Out_AV_Transfer )
   END_RUNG
   // the same network as SCL:
   #Out_AV_Transfer := #alwaysON AND #Actuator.AV_Transfer;
END_REGION

REGION Network 10: Pump Transfer
   RUNG wire#powerrail
      Contact( #alwaysON )
      wire#w1
      Contact( #State.Ready_For_Transfer )
      Move(in := #IN_Dose_Pump_Sp, out1 => #Out_P_Transfer_Sp)
   END_RUNG
   RUNG wire#w1
      Contact( #State.Ready_For_Transfer )
      Contact( #IN_Dose_Run )
      Contact( #IN_Dose_Pump_Cmd )
      Coil( #Actuator.P_Transfer )
   END_RUNG
   RUNG wire#w1
      Contact( #Actuator.P_Transfer )
      S_Coil( #Out_P_Transfer )
   END_RUNG
   RUNG wire#w1
      I_Contact( #Actuator.P_Transfer )
      I_Contact( #IN_FBCV )
      R_Coil( #Out_P_Transfer )
   END_RUNG
   // the same network as SCL:
   IF #alwaysON AND #State.Ready_For_Transfer THEN #Out_P_Transfer_Sp := #IN_Dose_Pump_Sp; END_IF;
   #Actuator.P_Transfer := #alwaysON AND #State.Ready_For_Transfer AND #IN_Dose_Run AND #IN_Dose_Pump_Cmd;
   IF #alwaysON AND #Actuator.P_Transfer THEN #Out_P_Transfer := TRUE; END_IF;
   IF #alwaysON AND NOT #Actuator.P_Transfer AND NOT #IN_FBCV THEN #Out_P_Transfer := FALSE; END_IF;
END_REGION

REGION Network 11: Control Valve
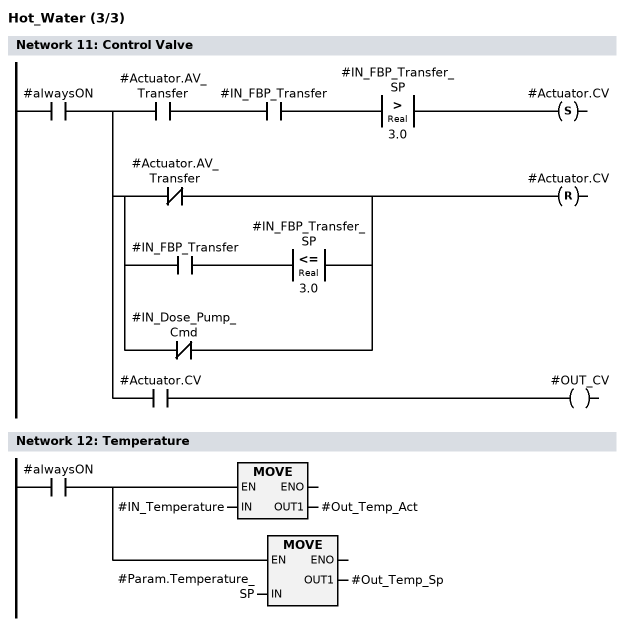
   RUNG wire#powerrail
      Contact( #alwaysON )
      wire#w1
      Contact( #Actuator.AV_Transfer )
      Contact( #IN_FBP_Transfer )
      { S7_Templates := "SrcType := Real" } GT_Contact(in1 := #IN_FBP_Transfer_SP, in2 := 3.0)
      S_Coil( #Actuator.CV )
   END_RUNG
   RUNG wire#w1
      I_Contact( #Actuator.AV_Transfer )
      wire#w2
      R_Coil( #Actuator.CV )
   END_RUNG
   RUNG wire#w1
      Contact( #IN_FBP_Transfer )
      { S7_Templates := "SrcType := Real" } LE_Contact(in1 := #IN_FBP_Transfer_SP, in2 := 3.0)
   END_RUNG wire#w2
   RUNG wire#w1
      I_Contact( #IN_Dose_Pump_Cmd )
   END_RUNG wire#w2
   RUNG wire#w1
      Contact( #Actuator.CV )
      Coil( #OUT_CV )
   END_RUNG
   // the same network as SCL:
   IF #alwaysON AND #Actuator.AV_Transfer AND #IN_FBP_Transfer AND (#IN_FBP_Transfer_SP > 3.0) THEN
       #Actuator.CV := TRUE;
   END_IF;
   IF #alwaysON AND (NOT #Actuator.AV_Transfer OR (#IN_FBP_Transfer AND (#IN_FBP_Transfer_SP <= 3.0)) OR NOT #IN_Dose_Pump_Cmd) THEN
       #Actuator.CV := FALSE;
   END_IF;
   #OUT_CV := #alwaysON AND #Actuator.CV;
END_REGION

REGION Network 12: Temperature
   RUNG wire#powerrail
      Contact( #alwaysON )
      wire#w1
      Move(in := #IN_Temperature, out1 => #Out_Temp_Act)
   END_RUNG
   RUNG wire#w1
      Move(in := #Param.Temperature_SP, out1 => #Out_Temp_Sp)
   END_RUNG
   // the same network as SCL:
   IF #alwaysON THEN
       #Out_Temp_Act := #IN_Temperature;
       #Out_Temp_Sp := #Param.Temperature_SP;
   END_IF;
END_REGION
END_FUNCTION_BLOCK

FUNCTION_BLOCK "IO Valve T02 Chili"   // FB302, LAD
{ S7_Optimized_Access := 'FALSE' }
VERSION : 0.1
// stored: AutoNumber false, IsIECCheckEnabled false, SetENOAutomatically false, UDAEnableTagReadback false
   VAR_INPUT
      lock : Bool;
      Init : Bool;
      testing : Bool;
      Reset : Bool;
   END_VAR
   VAR
      "AV-02.01" { S7_SetPoint := 'True'} : "Valve";   // AUTO BUTTERFLY VALVE INLET PROCESS WATER TO BFT CHILI AWETAN T-02.00
      "AV-02.02" { S7_SetPoint := 'True'} : "Valve";   // AUTO BUTTERFLY VALVE CIP SUPPLY TO BFT CHILI AWETAN T-02.00
      "AV-02.03" { S7_SetPoint := 'True'} : "Valve";   // AUTO BUTTERFLY VALVE OUTLET PRODUCT FROM BFT CHILI AWETAN T-02.00
      "AV-02.04" { S7_SetPoint := 'True'} : "Valve";   // AUTO BUTTERFLY VALVE OUTLET CIP TANK & LINE CHILI AWETAN T-02.00
      "AV-02.05" { S7_SetPoint := 'True'} : "Valve";   // AUTO BUTTERFLY VALVE DRAIN MONO PUMP P-02.01
      "AV-02.06" { S7_SetPoint := 'True'} : "Valve";
      "AV-02.07" { S7_SetPoint := 'True'} : "Valve";
      "AV-02.08" { S7_SetPoint := 'True'} : "Valve";
      "AV-02.09" { S7_SetPoint := 'True'} : "Valve";
      "AV-02.10" { S7_SetPoint := 'True'} : "Valve";
      "AV-02.11" { S7_SetPoint := 'True'} : "Valve";
      "AV-02.12" { S7_SetPoint := 'True'} : "Valve";
      "AV-02.13" { S7_SetPoint := 'True'} : "Valve";
      "AV-02.14" { S7_SetPoint := 'True'} : "Valve";
      "AV-02.15" { S7_SetPoint := 'True'} : "Valve";
      "AV-02.20" { S7_SetPoint := 'True'} : "Valve";
   END_VAR
BEGIN

REGION Network 1 (SCL): FB OPEN and CLOSE
   IF #testing THEN
       // Statement section IF
       #"AV-02.01".FB_OPEN := #"AV-02.01".QCMD_OP;
       #"AV-02.01".FB_CLOSE := NOT #"AV-02.01".QCMD_OP;
       #"AV-02.02".FB_OPEN := #"AV-02.02".QCMD_OP;
       #"AV-02.02".FB_CLOSE := NOT #"AV-02.02".QCMD_OP;
       #"AV-02.03".FB_OPEN := #"AV-02.03".QCMD_OP;
       #"AV-02.03".FB_CLOSE := NOT #"AV-02.03".QCMD_OP;
       #"AV-02.04".FB_OPEN := #"AV-02.04".QCMD_OP;
       #"AV-02.04".FB_CLOSE := NOT #"AV-02.04".QCMD_OP;
       #"AV-02.05".FB_OPEN := #"AV-02.05".QCMD_OP;
       #"AV-02.05".FB_CLOSE := NOT #"AV-02.05".QCMD_OP;
       #"AV-02.06".FB_OPEN := #"AV-02.06".QCMD_OP;
       #"AV-02.06".FB_CLOSE := NOT #"AV-02.06".QCMD_OP;
       #"AV-02.07".FB_OPEN := #"AV-02.07".QCMD_OP;
       #"AV-02.07".FB_CLOSE := NOT #"AV-02.07".QCMD_OP;
       #"AV-02.08".FB_OPEN := #"AV-02.08".QCMD_OP;
       #"AV-02.08".FB_CLOSE := NOT #"AV-02.08".QCMD_OP;
       #"AV-02.09".FB_OPEN := #"AV-02.09".QCMD_OP;
       #"AV-02.09".FB_CLOSE := NOT #"AV-02.09".QCMD_OP;
       #"AV-02.10".FB_OPEN := #"AV-02.10".QCMD_OP;
       #"AV-02.10".FB_CLOSE := NOT #"AV-02.10".QCMD_OP;
       #"AV-02.11".FB_OPEN := #"AV-02.11".QCMD_OP;
       #"AV-02.11".FB_CLOSE := NOT #"AV-02.11".QCMD_OP;
       #"AV-02.12".FB_OPEN := #"AV-02.12".QCMD_OP;
       #"AV-02.12".FB_CLOSE := NOT #"AV-02.12".QCMD_OP;
       #"AV-02.13".FB_OPEN := #"AV-02.13".QCMD_OP;
       #"AV-02.13".FB_CLOSE := NOT #"AV-02.13".QCMD_OP;
       #"AV-02.14".FB_OPEN := #"AV-02.14".QCMD_OP;
       #"AV-02.14".FB_CLOSE := NOT #"AV-02.14".QCMD_OP;
       #"AV-02.15".FB_OPEN := #"AV-02.15".QCMD_OP;
       #"AV-02.15".FB_CLOSE := NOT #"AV-02.15".QCMD_OP;
       #"AV-02.20".FB_OPEN := #"AV-02.20".QCMD_OP;
       #"AV-02.20".FB_CLOSE := NOT #"AV-02.20".QCMD_OP;
   ELSE
       // Statement section ELSE
       #"AV-02.01".FB_OPEN := NOT "ZSC-02.01";
       #"AV-02.01".FB_CLOSE := "ZSC-02.01";
       #"AV-02.02".FB_OPEN := NOT "ZSC-02.02";
       #"AV-02.02".FB_CLOSE := "ZSC-02.02";
       #"AV-02.03".FB_OPEN := NOT "ZSC-02.03";
       #"AV-02.03".FB_CLOSE := "ZSC-02.03";
       #"AV-02.04".FB_OPEN := NOT "ZSC-02.04";
       #"AV-02.04".FB_CLOSE := "ZSC-02.04";
       #"AV-02.05".FB_OPEN := #"AV-02.05".QCMD_OP;
       #"AV-02.05".FB_CLOSE := NOT #"AV-02.05".QCMD_OP;
       #"AV-02.06".FB_OPEN := #"AV-02.06".QCMD_OP;
       #"AV-02.06".FB_CLOSE := NOT #"AV-02.06".QCMD_OP;
       #"AV-02.07".FB_OPEN := #"AV-02.07".QCMD_OP;
       #"AV-02.07".FB_CLOSE := NOT #"AV-02.07".QCMD_OP;
       #"AV-02.08".FB_OPEN := #"AV-02.08".QCMD_OP;
       #"AV-02.08".FB_CLOSE := NOT #"AV-02.08".QCMD_OP;
       #"AV-02.09".FB_OPEN := #"AV-02.09".QCMD_OP;
       #"AV-02.09".FB_CLOSE := NOT #"AV-02.09".QCMD_OP;
       #"AV-02.10".FB_OPEN := #"AV-02.10".QCMD_OP;
       #"AV-02.10".FB_CLOSE := NOT #"AV-02.10".QCMD_OP;
       #"AV-02.11".FB_OPEN := NOT "ZSC-02.11";
       #"AV-02.11".FB_CLOSE := "ZSC-02.11";
       #"AV-02.12".FB_OPEN := NOT "ZSC-02.12";
       #"AV-02.12".FB_CLOSE := "ZSC-02.12";
       #"AV-02.13".FB_OPEN := NOT "ZSC-02.13";
       #"AV-02.13".FB_CLOSE := "ZSC-02.13";
       #"AV-02.14".FB_OPEN := #"AV-02.14".QCMD_OP;
       #"AV-02.14".FB_CLOSE := NOT #"AV-02.14".QCMD_OP;
       #"AV-02.15".FB_OPEN := #"AV-02.15".QCMD_OP;
       #"AV-02.15".FB_CLOSE := NOT #"AV-02.15".QCMD_OP;
       #"AV-02.20".FB_OPEN := #"AV-02.20".QCMD_OP;
       #"AV-02.20".FB_CLOSE := NOT #"AV-02.20".QCMD_OP;
   END_IF;
END_REGION

NETWORK
TITLE = FB Monitoring Time
// FB OPEN Time
      L     t#20s;
      T     #"AV-02.01".MON_T;
      T     #"AV-02.02".MON_T;
      T     #"AV-02.03".MON_T;
      T     #"AV-02.04".MON_T;
      T     #"AV-02.05".MON_T;
      T     #"AV-02.06".MON_T;
      T     #"AV-02.07".MON_T;
      T     #"AV-02.08".MON_T;
      T     #"AV-02.09".MON_T;
      T     #"AV-02.10".MON_T;
      T     #"AV-02.11".MON_T;
      T     #"AV-02.12".MON_T;
      T     #"AV-02.13".MON_T;
      T     #"AV-02.14".MON_T;
      T     #"AV-02.15".MON_T;
      T     #"AV-02.20".MON_T;
// FB CLOSE Time
      L     t#20s;
      T     #"AV-02.01".MON_T_CLOSE;
      T     #"AV-02.02".MON_T_CLOSE;
      T     #"AV-02.03".MON_T_CLOSE;
      T     #"AV-02.04".MON_T_CLOSE;
      T     #"AV-02.05".MON_T_CLOSE;
      T     #"AV-02.06".MON_T_CLOSE;
      T     #"AV-02.07".MON_T_CLOSE;
      T     #"AV-02.08".MON_T_CLOSE;
      T     #"AV-02.09".MON_T_CLOSE;
      T     #"AV-02.10".MON_T_CLOSE;
      T     #"AV-02.11".MON_T_CLOSE;
      T     #"AV-02.12".MON_T_CLOSE;
      T     #"AV-02.13".MON_T_CLOSE;
      T     #"AV-02.14".MON_T_CLOSE;
      T     #"AV-02.15".MON_T_CLOSE;
      T     #"AV-02.20".MON_T_CLOSE;

REGION Network 3: AV-02.01 w ZSC
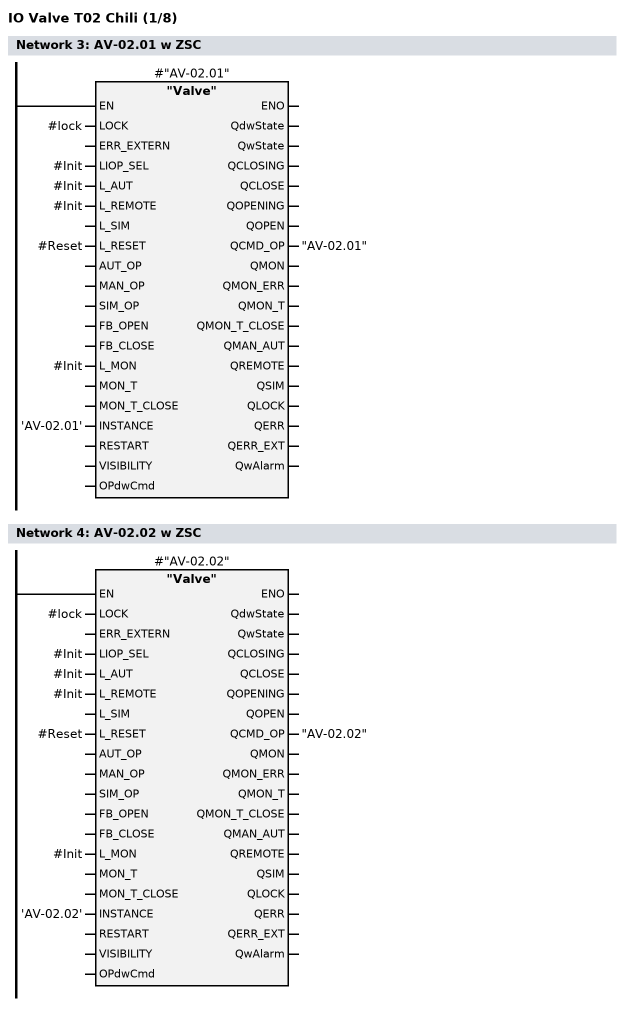
   RUNG wire#powerrail
      #"AV-02.01"(LOCK := #lock, ERR_EXTERN :=, LIOP_SEL := #Init, L_AUT := #Init, L_REMOTE := #Init, L_SIM :=, L_RESET := #Reset, AUT_OP :=, MAN_OP :=, SIM_OP :=, FB_OPEN :=, FB_CLOSE :=, L_MON := #Init, MON_T :=, MON_T_CLOSE :=, INSTANCE := 'AV-02.01', RESTART :=, VISIBILITY :=, OPdwCmd :=, QdwState =>, QwState =>, QCLOSING =>, QCLOSE =>, QOPENING =>, QOPEN =>, QCMD_OP => "AV-02.01", QMON =>, QMON_ERR =>, QMON_T =>, QMON_T_CLOSE =>, QMAN_AUT =>, QREMOTE =>, QSIM =>, QLOCK =>, QERR =>, QERR_EXT =>, QwAlarm =>)
   END_RUNG
   // the same network as SCL:
   #"AV-02.01"(LOCK := #lock,   // "Valve"
               LIOP_SEL := #Init,
               L_AUT := #Init,
               L_REMOTE := #Init,
               L_RESET := #Reset,
               L_MON := #Init,
               INSTANCE := 'AV-02.01',
               QCMD_OP => "AV-02.01");
END_REGION

REGION Network 4: AV-02.02 w ZSC
   RUNG wire#powerrail
      #"AV-02.02"(LOCK := #lock, ERR_EXTERN :=, LIOP_SEL := #Init, L_AUT := #Init, L_REMOTE := #Init, L_SIM :=, L_RESET := #Reset, AUT_OP :=, MAN_OP :=, SIM_OP :=, FB_OPEN :=, FB_CLOSE :=, L_MON := #Init, MON_T :=, MON_T_CLOSE :=, INSTANCE := 'AV-02.02', RESTART :=, VISIBILITY :=, OPdwCmd :=, QdwState =>, QwState =>, QCLOSING =>, QCLOSE =>, QOPENING =>, QOPEN =>, QCMD_OP => "AV-02.02", QMON =>, QMON_ERR =>, QMON_T =>, QMON_T_CLOSE =>, QMAN_AUT =>, QREMOTE =>, QSIM =>, QLOCK =>, QERR =>, QERR_EXT =>, QwAlarm =>)
   END_RUNG
   // the same network as SCL:
   #"AV-02.02"(LOCK := #lock,   // "Valve"
               LIOP_SEL := #Init,
               L_AUT := #Init,
               L_REMOTE := #Init,
               L_RESET := #Reset,
               L_MON := #Init,
               INSTANCE := 'AV-02.02',
               QCMD_OP => "AV-02.02");
END_REGION

REGION Network 5: AV-02.03 w ZSC
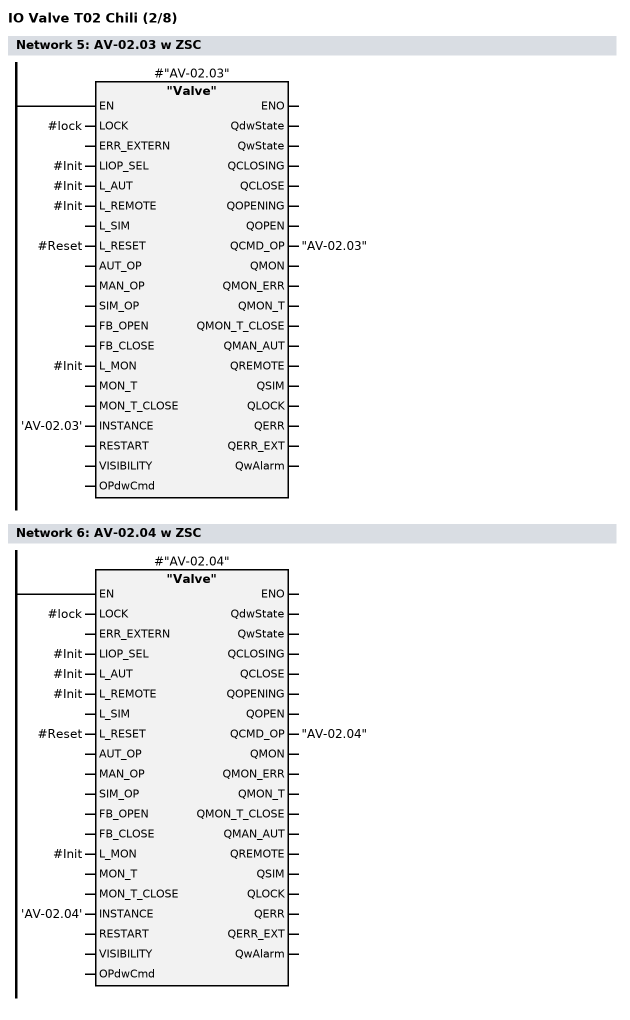
   RUNG wire#powerrail
      #"AV-02.03"(LOCK := #lock, ERR_EXTERN :=, LIOP_SEL := #Init, L_AUT := #Init, L_REMOTE := #Init, L_SIM :=, L_RESET := #Reset, AUT_OP :=, MAN_OP :=, SIM_OP :=, FB_OPEN :=, FB_CLOSE :=, L_MON := #Init, MON_T :=, MON_T_CLOSE :=, INSTANCE := 'AV-02.03', RESTART :=, VISIBILITY :=, OPdwCmd :=, QdwState =>, QwState =>, QCLOSING =>, QCLOSE =>, QOPENING =>, QOPEN =>, QCMD_OP => "AV-02.03", QMON =>, QMON_ERR =>, QMON_T =>, QMON_T_CLOSE =>, QMAN_AUT =>, QREMOTE =>, QSIM =>, QLOCK =>, QERR =>, QERR_EXT =>, QwAlarm =>)
   END_RUNG
   // the same network as SCL:
   #"AV-02.03"(LOCK := #lock,   // "Valve"
               LIOP_SEL := #Init,
               L_AUT := #Init,
               L_REMOTE := #Init,
               L_RESET := #Reset,
               L_MON := #Init,
               INSTANCE := 'AV-02.03',
               QCMD_OP => "AV-02.03");
END_REGION

REGION Network 6: AV-02.04 w ZSC
   RUNG wire#powerrail
      #"AV-02.04"(LOCK := #lock, ERR_EXTERN :=, LIOP_SEL := #Init, L_AUT := #Init, L_REMOTE := #Init, L_SIM :=, L_RESET := #Reset, AUT_OP :=, MAN_OP :=, SIM_OP :=, FB_OPEN :=, FB_CLOSE :=, L_MON := #Init, MON_T :=, MON_T_CLOSE :=, INSTANCE := 'AV-02.04', RESTART :=, VISIBILITY :=, OPdwCmd :=, QdwState =>, QwState =>, QCLOSING =>, QCLOSE =>, QOPENING =>, QOPEN =>, QCMD_OP => "AV-02.04", QMON =>, QMON_ERR =>, QMON_T =>, QMON_T_CLOSE =>, QMAN_AUT =>, QREMOTE =>, QSIM =>, QLOCK =>, QERR =>, QERR_EXT =>, QwAlarm =>)
   END_RUNG
   // the same network as SCL:
   #"AV-02.04"(LOCK := #lock,   // "Valve"
               LIOP_SEL := #Init,
               L_AUT := #Init,
               L_REMOTE := #Init,
               L_RESET := #Reset,
               L_MON := #Init,
               INSTANCE := 'AV-02.04',
               QCMD_OP => "AV-02.04");
END_REGION

REGION Network 7: AV-02.05
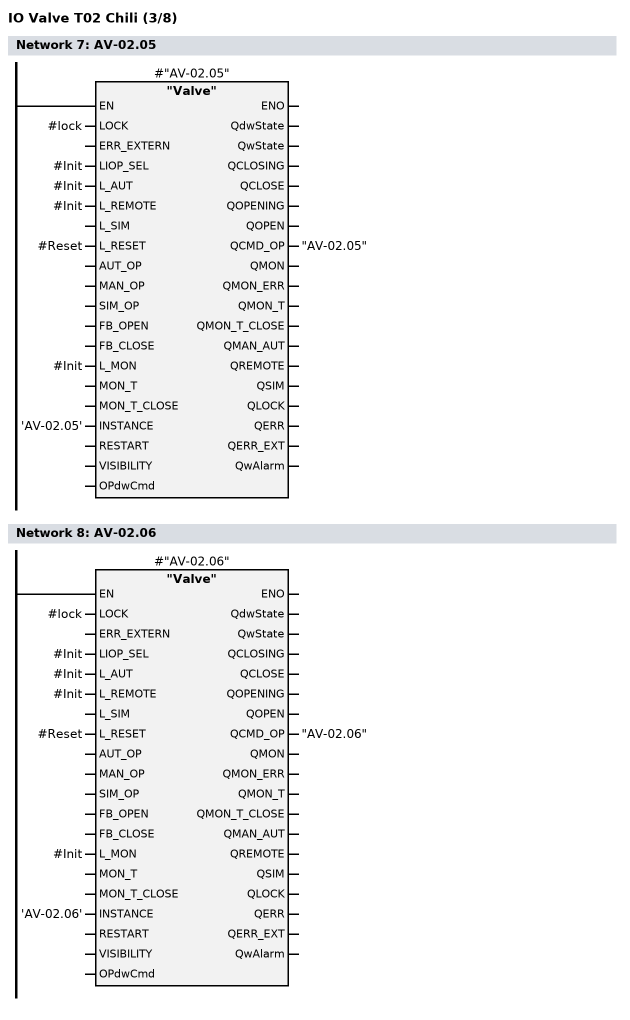
   RUNG wire#powerrail
      #"AV-02.05"(LOCK := #lock, ERR_EXTERN :=, LIOP_SEL := #Init, L_AUT := #Init, L_REMOTE := #Init, L_SIM :=, L_RESET := #Reset, AUT_OP :=, MAN_OP :=, SIM_OP :=, FB_OPEN :=, FB_CLOSE :=, L_MON := #Init, MON_T :=, MON_T_CLOSE :=, INSTANCE := 'AV-02.05', RESTART :=, VISIBILITY :=, OPdwCmd :=, QdwState =>, QwState =>, QCLOSING =>, QCLOSE =>, QOPENING =>, QOPEN =>, QCMD_OP => "AV-02.05", QMON =>, QMON_ERR =>, QMON_T =>, QMON_T_CLOSE =>, QMAN_AUT =>, QREMOTE =>, QSIM =>, QLOCK =>, QERR =>, QERR_EXT =>, QwAlarm =>)
   END_RUNG
   // the same network as SCL:
   #"AV-02.05"(LOCK := #lock,   // "Valve"
               LIOP_SEL := #Init,
               L_AUT := #Init,
               L_REMOTE := #Init,
               L_RESET := #Reset,
               L_MON := #Init,
               INSTANCE := 'AV-02.05',
               QCMD_OP => "AV-02.05");
END_REGION

REGION Network 8: AV-02.06
   RUNG wire#powerrail
      #"AV-02.06"(LOCK := #lock, ERR_EXTERN :=, LIOP_SEL := #Init, L_AUT := #Init, L_REMOTE := #Init, L_SIM :=, L_RESET := #Reset, AUT_OP :=, MAN_OP :=, SIM_OP :=, FB_OPEN :=, FB_CLOSE :=, L_MON := #Init, MON_T :=, MON_T_CLOSE :=, INSTANCE := 'AV-02.06', RESTART :=, VISIBILITY :=, OPdwCmd :=, QdwState =>, QwState =>, QCLOSING =>, QCLOSE =>, QOPENING =>, QOPEN =>, QCMD_OP => "AV-02.06", QMON =>, QMON_ERR =>, QMON_T =>, QMON_T_CLOSE =>, QMAN_AUT =>, QREMOTE =>, QSIM =>, QLOCK =>, QERR =>, QERR_EXT =>, QwAlarm =>)
   END_RUNG
   // the same network as SCL:
   #"AV-02.06"(LOCK := #lock,   // "Valve"
               LIOP_SEL := #Init,
               L_AUT := #Init,
               L_REMOTE := #Init,
               L_RESET := #Reset,
               L_MON := #Init,
               INSTANCE := 'AV-02.06',
               QCMD_OP => "AV-02.06");
END_REGION

REGION Network 9: AV-02.07
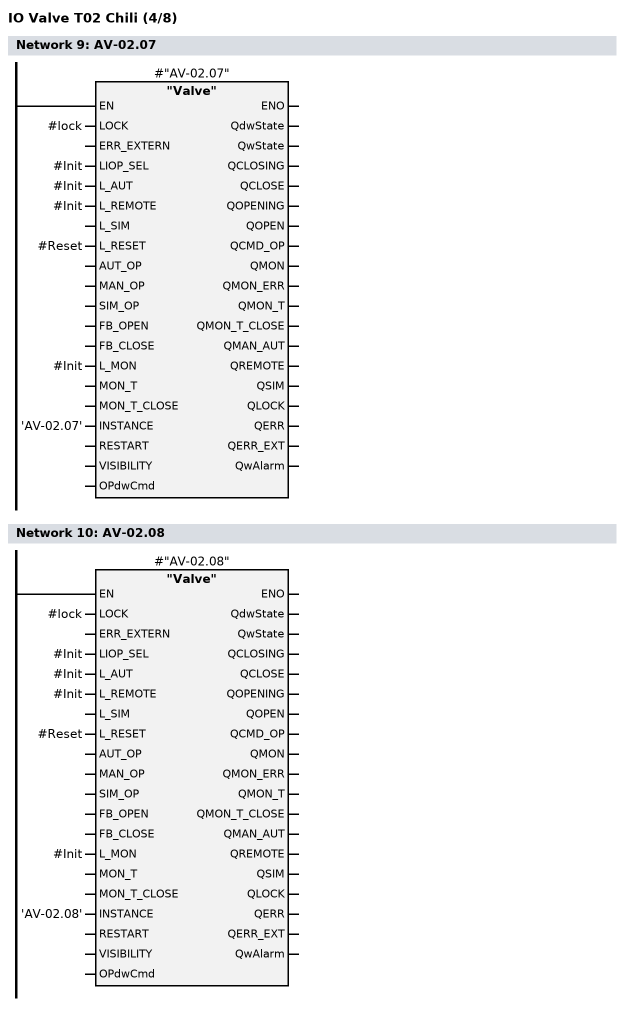
   RUNG wire#powerrail
      #"AV-02.07"(LOCK := #lock, ERR_EXTERN :=, LIOP_SEL := #Init, L_AUT := #Init, L_REMOTE := #Init, L_SIM :=, L_RESET := #Reset, AUT_OP :=, MAN_OP :=, SIM_OP :=, FB_OPEN :=, FB_CLOSE :=, L_MON := #Init, MON_T :=, MON_T_CLOSE :=, INSTANCE := 'AV-02.07', RESTART :=, VISIBILITY :=, OPdwCmd :=, QdwState =>, QwState =>, QCLOSING =>, QCLOSE =>, QOPENING =>, QOPEN =>, QCMD_OP =>, QMON =>, QMON_ERR =>, QMON_T =>, QMON_T_CLOSE =>, QMAN_AUT =>, QREMOTE =>, QSIM =>, QLOCK =>, QERR =>, QERR_EXT =>, QwAlarm =>)
   END_RUNG
   // the same network as SCL:
   #"AV-02.07"(LOCK := #lock,   // "Valve"
               LIOP_SEL := #Init,
               L_AUT := #Init,
               L_REMOTE := #Init,
               L_RESET := #Reset,
               L_MON := #Init,
               INSTANCE := 'AV-02.07');
END_REGION

REGION Network 10: AV-02.08
   RUNG wire#powerrail
      #"AV-02.08"(LOCK := #lock, ERR_EXTERN :=, LIOP_SEL := #Init, L_AUT := #Init, L_REMOTE := #Init, L_SIM :=, L_RESET := #Reset, AUT_OP :=, MAN_OP :=, SIM_OP :=, FB_OPEN :=, FB_CLOSE :=, L_MON := #Init, MON_T :=, MON_T_CLOSE :=, INSTANCE := 'AV-02.08', RESTART :=, VISIBILITY :=, OPdwCmd :=, QdwState =>, QwState =>, QCLOSING =>, QCLOSE =>, QOPENING =>, QOPEN =>, QCMD_OP =>, QMON =>, QMON_ERR =>, QMON_T =>, QMON_T_CLOSE =>, QMAN_AUT =>, QREMOTE =>, QSIM =>, QLOCK =>, QERR =>, QERR_EXT =>, QwAlarm =>)
   END_RUNG
   // the same network as SCL:
   #"AV-02.08"(LOCK := #lock,   // "Valve"
               LIOP_SEL := #Init,
               L_AUT := #Init,
               L_REMOTE := #Init,
               L_RESET := #Reset,
               L_MON := #Init,
               INSTANCE := 'AV-02.08');
END_REGION

REGION Network 11: AV-02.09
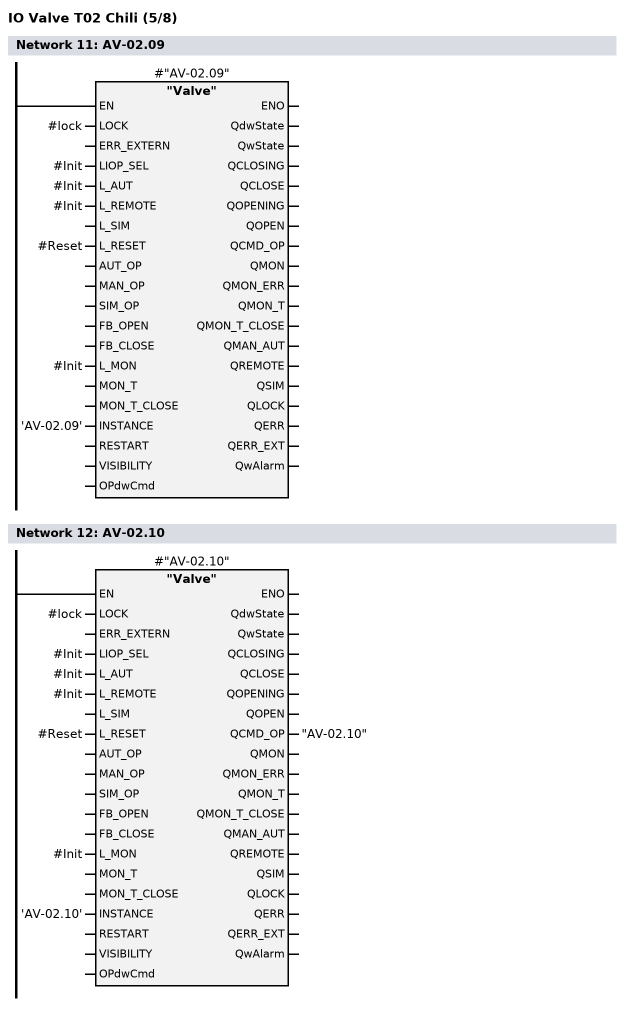
   RUNG wire#powerrail
      #"AV-02.09"(LOCK := #lock, ERR_EXTERN :=, LIOP_SEL := #Init, L_AUT := #Init, L_REMOTE := #Init, L_SIM :=, L_RESET := #Reset, AUT_OP :=, MAN_OP :=, SIM_OP :=, FB_OPEN :=, FB_CLOSE :=, L_MON := #Init, MON_T :=, MON_T_CLOSE :=, INSTANCE := 'AV-02.09', RESTART :=, VISIBILITY :=, OPdwCmd :=, QdwState =>, QwState =>, QCLOSING =>, QCLOSE =>, QOPENING =>, QOPEN =>, QCMD_OP =>, QMON =>, QMON_ERR =>, QMON_T =>, QMON_T_CLOSE =>, QMAN_AUT =>, QREMOTE =>, QSIM =>, QLOCK =>, QERR =>, QERR_EXT =>, QwAlarm =>)
   END_RUNG
   // the same network as SCL:
   #"AV-02.09"(LOCK := #lock,   // "Valve"
               LIOP_SEL := #Init,
               L_AUT := #Init,
               L_REMOTE := #Init,
               L_RESET := #Reset,
               L_MON := #Init,
               INSTANCE := 'AV-02.09');
END_REGION

REGION Network 12: AV-02.10
   RUNG wire#powerrail
      #"AV-02.10"(LOCK := #lock, ERR_EXTERN :=, LIOP_SEL := #Init, L_AUT := #Init, L_REMOTE := #Init, L_SIM :=, L_RESET := #Reset, AUT_OP :=, MAN_OP :=, SIM_OP :=, FB_OPEN :=, FB_CLOSE :=, L_MON := #Init, MON_T :=, MON_T_CLOSE :=, INSTANCE := 'AV-02.10', RESTART :=, VISIBILITY :=, OPdwCmd :=, QdwState =>, QwState =>, QCLOSING =>, QCLOSE =>, QOPENING =>, QOPEN =>, QCMD_OP => "AV-02.10", QMON =>, QMON_ERR =>, QMON_T =>, QMON_T_CLOSE =>, QMAN_AUT =>, QREMOTE =>, QSIM =>, QLOCK =>, QERR =>, QERR_EXT =>, QwAlarm =>)
   END_RUNG
   // the same network as SCL:
   #"AV-02.10"(LOCK := #lock,   // "Valve"
               LIOP_SEL := #Init,
               L_AUT := #Init,
               L_REMOTE := #Init,
               L_RESET := #Reset,
               L_MON := #Init,
               INSTANCE := 'AV-02.10',
               QCMD_OP => "AV-02.10");
END_REGION

REGION Network 13: AV-02.11 w ZSC
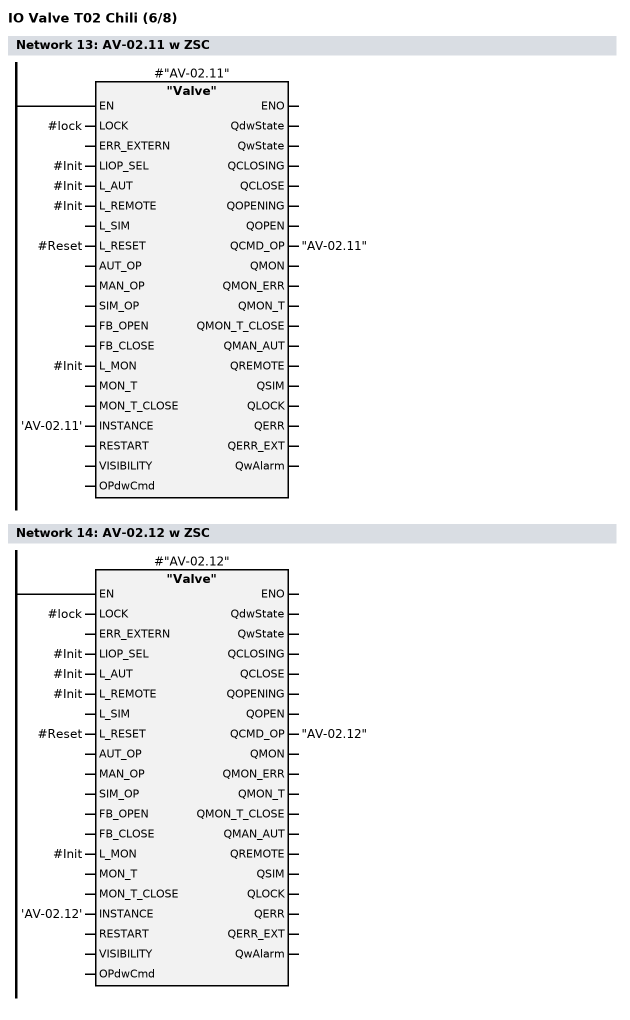
   RUNG wire#powerrail
      #"AV-02.11"(LOCK := #lock, ERR_EXTERN :=, LIOP_SEL := #Init, L_AUT := #Init, L_REMOTE := #Init, L_SIM :=, L_RESET := #Reset, AUT_OP :=, MAN_OP :=, SIM_OP :=, FB_OPEN :=, FB_CLOSE :=, L_MON := #Init, MON_T :=, MON_T_CLOSE :=, INSTANCE := 'AV-02.11', RESTART :=, VISIBILITY :=, OPdwCmd :=, QdwState =>, QwState =>, QCLOSING =>, QCLOSE =>, QOPENING =>, QOPEN =>, QCMD_OP => "AV-02.11", QMON =>, QMON_ERR =>, QMON_T =>, QMON_T_CLOSE =>, QMAN_AUT =>, QREMOTE =>, QSIM =>, QLOCK =>, QERR =>, QERR_EXT =>, QwAlarm =>)
   END_RUNG
   // the same network as SCL:
   #"AV-02.11"(LOCK := #lock,   // "Valve"
               LIOP_SEL := #Init,
               L_AUT := #Init,
               L_REMOTE := #Init,
               L_RESET := #Reset,
               L_MON := #Init,
               INSTANCE := 'AV-02.11',
               QCMD_OP => "AV-02.11");
END_REGION

REGION Network 14: AV-02.12 w ZSC
   RUNG wire#powerrail
      #"AV-02.12"(LOCK := #lock, ERR_EXTERN :=, LIOP_SEL := #Init, L_AUT := #Init, L_REMOTE := #Init, L_SIM :=, L_RESET := #Reset, AUT_OP :=, MAN_OP :=, SIM_OP :=, FB_OPEN :=, FB_CLOSE :=, L_MON := #Init, MON_T :=, MON_T_CLOSE :=, INSTANCE := 'AV-02.12', RESTART :=, VISIBILITY :=, OPdwCmd :=, QdwState =>, QwState =>, QCLOSING =>, QCLOSE =>, QOPENING =>, QOPEN =>, QCMD_OP => "AV-02.12", QMON =>, QMON_ERR =>, QMON_T =>, QMON_T_CLOSE =>, QMAN_AUT =>, QREMOTE =>, QSIM =>, QLOCK =>, QERR =>, QERR_EXT =>, QwAlarm =>)
   END_RUNG
   // the same network as SCL:
   #"AV-02.12"(LOCK := #lock,   // "Valve"
               LIOP_SEL := #Init,
               L_AUT := #Init,
               L_REMOTE := #Init,
               L_RESET := #Reset,
               L_MON := #Init,
               INSTANCE := 'AV-02.12',
               QCMD_OP => "AV-02.12");
END_REGION

REGION Network 15: AV-02.13 w ZSC
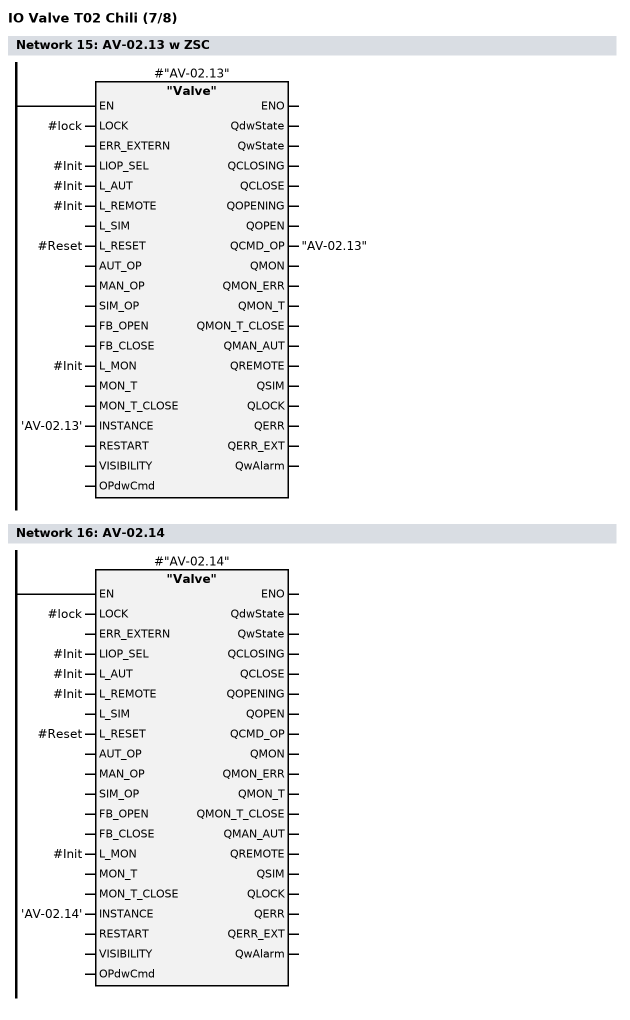
   RUNG wire#powerrail
      #"AV-02.13"(LOCK := #lock, ERR_EXTERN :=, LIOP_SEL := #Init, L_AUT := #Init, L_REMOTE := #Init, L_SIM :=, L_RESET := #Reset, AUT_OP :=, MAN_OP :=, SIM_OP :=, FB_OPEN :=, FB_CLOSE :=, L_MON := #Init, MON_T :=, MON_T_CLOSE :=, INSTANCE := 'AV-02.13', RESTART :=, VISIBILITY :=, OPdwCmd :=, QdwState =>, QwState =>, QCLOSING =>, QCLOSE =>, QOPENING =>, QOPEN =>, QCMD_OP => "AV-02.13", QMON =>, QMON_ERR =>, QMON_T =>, QMON_T_CLOSE =>, QMAN_AUT =>, QREMOTE =>, QSIM =>, QLOCK =>, QERR =>, QERR_EXT =>, QwAlarm =>)
   END_RUNG
   // the same network as SCL:
   #"AV-02.13"(LOCK := #lock,   // "Valve"
               LIOP_SEL := #Init,
               L_AUT := #Init,
               L_REMOTE := #Init,
               L_RESET := #Reset,
               L_MON := #Init,
               INSTANCE := 'AV-02.13',
               QCMD_OP => "AV-02.13");
END_REGION

REGION Network 16: AV-02.14
   RUNG wire#powerrail
      #"AV-02.14"(LOCK := #lock, ERR_EXTERN :=, LIOP_SEL := #Init, L_AUT := #Init, L_REMOTE := #Init, L_SIM :=, L_RESET := #Reset, AUT_OP :=, MAN_OP :=, SIM_OP :=, FB_OPEN :=, FB_CLOSE :=, L_MON := #Init, MON_T :=, MON_T_CLOSE :=, INSTANCE := 'AV-02.14', RESTART :=, VISIBILITY :=, OPdwCmd :=, QdwState =>, QwState =>, QCLOSING =>, QCLOSE =>, QOPENING =>, QOPEN =>, QCMD_OP =>, QMON =>, QMON_ERR =>, QMON_T =>, QMON_T_CLOSE =>, QMAN_AUT =>, QREMOTE =>, QSIM =>, QLOCK =>, QERR =>, QERR_EXT =>, QwAlarm =>)
   END_RUNG
   // the same network as SCL:
   #"AV-02.14"(LOCK := #lock,   // "Valve"
               LIOP_SEL := #Init,
               L_AUT := #Init,
               L_REMOTE := #Init,
               L_RESET := #Reset,
               L_MON := #Init,
               INSTANCE := 'AV-02.14');
END_REGION

REGION Network 17: AV-02.15
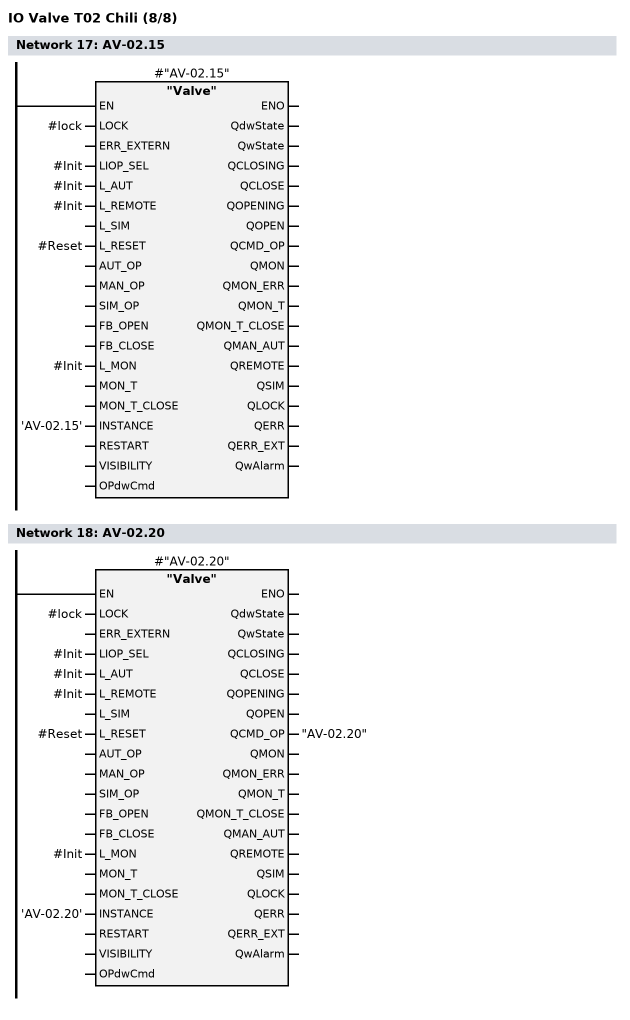
   RUNG wire#powerrail
      #"AV-02.15"(LOCK := #lock, ERR_EXTERN :=, LIOP_SEL := #Init, L_AUT := #Init, L_REMOTE := #Init, L_SIM :=, L_RESET := #Reset, AUT_OP :=, MAN_OP :=, SIM_OP :=, FB_OPEN :=, FB_CLOSE :=, L_MON := #Init, MON_T :=, MON_T_CLOSE :=, INSTANCE := 'AV-02.15', RESTART :=, VISIBILITY :=, OPdwCmd :=, QdwState =>, QwState =>, QCLOSING =>, QCLOSE =>, QOPENING =>, QOPEN =>, QCMD_OP =>, QMON =>, QMON_ERR =>, QMON_T =>, QMON_T_CLOSE =>, QMAN_AUT =>, QREMOTE =>, QSIM =>, QLOCK =>, QERR =>, QERR_EXT =>, QwAlarm =>)
   END_RUNG
   // the same network as SCL:
   #"AV-02.15"(LOCK := #lock,   // "Valve"
               LIOP_SEL := #Init,
               L_AUT := #Init,
               L_REMOTE := #Init,
               L_RESET := #Reset,
               L_MON := #Init,
               INSTANCE := 'AV-02.15');
END_REGION

REGION Network 18: AV-02.20
   RUNG wire#powerrail
      #"AV-02.20"(LOCK := #lock, ERR_EXTERN :=, LIOP_SEL := #Init, L_AUT := #Init, L_REMOTE := #Init, L_SIM :=, L_RESET := #Reset, AUT_OP :=, MAN_OP :=, SIM_OP :=, FB_OPEN :=, FB_CLOSE :=, L_MON := #Init, MON_T :=, MON_T_CLOSE :=, INSTANCE := 'AV-02.20', RESTART :=, VISIBILITY :=, OPdwCmd :=, QdwState =>, QwState =>, QCLOSING =>, QCLOSE =>, QOPENING =>, QOPEN =>, QCMD_OP => "AV-02.20", QMON =>, QMON_ERR =>, QMON_T =>, QMON_T_CLOSE =>, QMAN_AUT =>, QREMOTE =>, QSIM =>, QLOCK =>, QERR =>, QERR_EXT =>, QwAlarm =>)
   END_RUNG
   // the same network as SCL:
   #"AV-02.20"(LOCK := #lock,   // "Valve"
               LIOP_SEL := #Init,
               L_AUT := #Init,
               L_REMOTE := #Init,
               L_RESET := #Reset,
               L_MON := #Init,
               INSTANCE := 'AV-02.20',
               QCMD_OP => "AV-02.20");
END_REGION
END_FUNCTION_BLOCK

FUNCTION_BLOCK "Valve"
{ S7_Optimized_Access := 'FALSE' }
VERSION : 0.1
   VAR_INPUT 
      LOCK : Bool;   // 1 = Interlock active
      ERR_EXTERN : Bool;   // 1 = External error arised
      LIOP_SEL : Bool;   // 0 = Operator; 1 = Linking
      L_AUT : Bool;   // 0 = Manual; 1 = Automatic
      L_REMOTE : Bool;   // 0 = Local; 1 = Remote
      L_SIM : Bool;   // 0 = Normal; 1 = Simulation
      L_RESET : Bool;   // 1 = Reset error peripherie
      AUT_OP : Bool;   // 1 = CMD OPEN Automatic
      MAN_OP : Bool;   // 1 = CMD OPEN Manual
      SIM_OP : Bool;   // 1 = CMD OPEN Simulation
      FB_OPEN : Bool;   // 1 = Feedback valve OPEN
      FB_CLOSE : Bool;   // 1 = Feedback valve CLOSED
      L_MON : Bool;   // 1 = Monitoring OPEN
      MON_T : Time := t#5s;   // Monitoring opening time in process mode
      MON_T_CLOSE : Time := t#5s;   // Monitoring closing time in process mode
      INSTANCE : String := 'Valve_001';   // Filter attribute for message view, also used for labelling
      RESTART : Bool;   // 1 = Initialize FB at startup (first cycle of PLC)
   END_VAR

   VAR_OUTPUT 
      QdwState : DWord;   // Status HMI
      QwState : Int;   // Valve: 0 = Close; 1 = Opening; 2 = Open; 3 = Closing
      QCLOSING : Bool;   // 1 = Closing
      QCLOSE : Bool;   // 1 = Close
      QOPENING : Bool;   // 1 = Opening
      QOPEN : Bool;   // 1 = Open
      QCMD_OP : Bool;   // 0 = Close; 1 = Open (automatic & manual mode)
      QMON : Bool;   // 1 = Monitoring is ON
      QMON_ERR : Bool;   // 1 = Monitoring errror
      QMON_T : Time;   // Expierd opening time in process mode
      QMON_T_CLOSE : Time;   // Expierd closing time in process mode
      QMAN_AUT : Bool;   // 0 = Manual; 1 = Automatic
      QREMOTE : Bool;   // 0 = Local; 1 = Remote
      QSIM : Bool;   // 0 = Normal; 1 = Simulation
      QLOCK : Bool;   // 1 = Interlock is active
      QERR : Bool;   // 1 = Common error
      QERR_EXT : Bool;   // 1 = External error
      QwAlarm : Word;   // Bit alarm procedure
   END_VAR

   VAR_IN_OUT 
      VISIBILITY : Byte;   // Bit 0: Tab1 of window; Bit 1: Tab2 of window; ... ; Bit 7: Minimize
      OPdwCmd : DWord;   // Contorl word HMI
   END_VAR

   VAR 
      OP_RESET : Bool;   // Reset errors
      FB_SIM_OPEN : Bool;   // 1 = Feedback Valve is OPEN in simulation mode
      FB_SIM_CLOSE : Bool;   // 1 = Feedback Valve is CLOSE in simulation mode
      SIM_T : Time := t#5s;   // Monitoring opening time in simulation mode
      QSIM_T : Time;   // Remaining opening time in simulation mode
      SIM_T_CLOSE : Time := T#5s;   // Monitoring closing time in simulation mode
      QSIM_T_CLOSE : Time;   // Remaining closing time in simulation mode
      QCMD_SIM : Bool;   // 0 = Close; 1 = Open (simulation mode)
      OP_VISIBILITY : Byte;   // Bit 0: Tab1 of window; Bit 1: Tab2 of window; ... ; Bit 7: Minimize
      VISIBILITY_OLD : Byte;   // Save last status of VISIBILITY
      SE_L_RESET_LINK : Bool;   // Signal edge for the reset input from linking
      SE_L_RESET_LINK_COND : Bool;   // Condition of signal edge
      SE_L_RESET_OP : Bool;   // Signal edge for the reset input from operator
      TOPENING {InstructionName := 'TON_TIME'; LibVersion := '1.0'} : TON_TIME;   // Maximum opening time
      TCLOSING {InstructionName := 'TON_TIME'; LibVersion := '1.0'} : TON_TIME;
      TOPENING_SIM {InstructionName := 'TON_TIME'; LibVersion := '1.0'} : TON_TIME;
      TCLOSING_SIM {InstructionName := 'TON_TIME'; LibVersion := '1.0'} : TON_TIME;
   END_VAR

   VAR_TEMP 
      CON_ERR : Bool;   // Error in valve condition
      MON_ERR_OPENING : Bool;   // Monitoring error for opening valve in process mode
      MON_ERR_CLOSING : Bool;   // Monitoring error for closing valve in process mode
      MON_SIM_OPENING : Bool;   // Monitoring error for opening valve in simulation mode
      MON_SIM_CLOSING : Bool;   // Monitoring error for closing valve in simulation mode
      FB_ERR : Bool;   // Feedback error in process mode
   END_VAR


BEGIN
	(********************************
	           Start up
	*********************************)
	IF #RESTART= true THEN
	  // Restart case
	  #QCMD_OP:= false;
	  #QCLOSE:=true;
	  #QOPENING:=false;
	  #QOPEN:=false;
	  #QCLOSING:=false;
	  #VISIBILITY:=0;
	  #OPdwCmd:=0;
	ELSE
	  // Normal case
	  
	 (******************************************
	    Network 1: Operating mode: manual/automatic
	    Vaiable: OPdwCmd  Bit:  16  =  Manual
	    Vaiable: OPdwCmd  Bit:  17  =  Automatic
	  *******************************************)
	  IF (#LIOP_SEL=true AND #L_AUT=true) OR (#OPdwCmd.%X17=true AND #LIOP_SEL=false) THEN
	    #QMAN_AUT:=true;
	    #OPdwCmd.%X16:=false;
	    #OPdwCmd.%X17:=false;
	  ELSIF (#LIOP_SEL=true AND #L_AUT=false) OR (#OPdwCmd.%X16=true AND #LIOP_SEL=false) THEN
	    #QMAN_AUT:= false;
	    #OPdwCmd.%X16:=false;
	    #OPdwCmd.%X17:=false;
	  END_IF;
	  
	  (******************************************
	    Network 2: Control mode: local/remote
	    Vaiable: OPdwCmd  Bit:  18  =  Local
	    Vaiable: OPdwCmd  Bit:  19  =  Remote
	  *******************************************)
	  IF (#LIOP_SEL=true AND #L_REMOTE=true) OR (#OPdwCmd.%X19=true AND #LIOP_SEL=false) THEN
	    #QREMOTE:=true;
	    #OPdwCmd.%X18:=false;
	    #OPdwCmd.%X19:=false;
	  ELSIF (#LIOP_SEL=true AND #L_REMOTE=false) OR (#OPdwCmd.%X18=true AND #LIOP_SEL=false) THEN
	    #QREMOTE:= false;
	    #OPdwCmd.%X18:=false;
	    #OPdwCmd.%X19:=false;
	  END_IF;
	  
	  (******************************************
	    Network 3: Simulation On/Off
	    Vaiable: OPdwCmd  Bit:  20  =  Process
	    Vaiable: OPdwCmd  Bit:  21  =  Simulation
	  *******************************************)
	  IF (#LIOP_SEL=true AND #L_SIM=true) OR (#OPdwCmd.%X21=true AND #LIOP_SEL=false) THEN
	    #QSIM:=true;
	    #OPdwCmd.%X20:=false;
	    #OPdwCmd.%X21:=false;
	  ELSIF (#LIOP_SEL=true AND #L_SIM=false) OR (#OPdwCmd.%X20=true AND #LIOP_SEL=false) THEN
	    #QSIM:= false;
	    #OPdwCmd.%X20:=false;
	    #OPdwCmd.%X21:=false;
	  END_IF;
	  
	  (*************************************
	    Network 4: Reset Operation
	    Vaiable: OPdwCmd  Bit:  24  =  Reset
	  **************************************)
	  // Rising edge by linking
	  IF #L_RESET=true AND #SE_L_RESET_LINK_COND=false THEN
	    #SE_L_RESET_LINK:=true;
	    #SE_L_RESET_LINK_COND:=true;
	  ELSIF #L_RESET=true AND #SE_L_RESET_LINK_COND=true THEN
	    #SE_L_RESET_LINK:=false;
	  ELSE
	    #SE_L_RESET_LINK_COND:=false;
	  END_IF;
	  // Rising edge by operator
	  IF #OPdwCmd.%X24=true THEN
	    #SE_L_RESET_OP:=true;
	    #OPdwCmd.%X24:=false;
	  ELSE
	    #SE_L_RESET_OP:=false;
	  END_IF;
	  // Reset error
	  #OP_RESET:=(#SE_L_RESET_LINK OR (#SE_L_RESET_OP AND NOT #LIOP_SEL)) AND NOT #LOCK;
	  
	  (**********************************************
	    Network 5: Monitoring feedback ON/OFF
	    Vaiable: OPdwCmd  Bit:  8  =  Monitoring ON
	    Vaiable: OPdwCmd  Bit:  9  =  Monitoring OFF
	  ***********************************************)
	  IF (#LIOP_SEL=true AND #L_MON=false) OR (#OPdwCmd.%X9=true AND #LIOP_SEL=false)THEN
	    #QMON:=false;
	    #OPdwCmd.%X8:=false;
	    #OPdwCmd.%X9:=false;
	  ELSIF (#LIOP_SEL=true AND #L_MON=true) OR (#OPdwCmd.%X8=true AND #LIOP_SEL=false)THEN
	    #QMON:=true;
	    #OPdwCmd.%X8:=false;
	    #OPdwCmd.%X9:=false;
	  END_IF;
	
	  (**********************************************
	    Network 6: OPEN/CLOSE Valve
	    Vaiable: OPdwCmd  Bit:  0  =  OPEN Valve
	    Vaiable: OPdwCmd  Bit:  1  =  CLOSE Valve
	  ***********************************************)
	  IF #QERR=false THEN
	    // No errors occurs
	    IF #QSIM=false THEN
	     // Simulation mode is not active
	      // Automatic/Manual mode
	      IF #QMAN_AUT=true THEN
	        // Automatic mode is active
	        // OPEN/CLOSE valve by linking (AUT_OP)
	        #QCMD_OP:=#AUT_OP;
	      ELSE
	       // Automatic mode is not active
	        // Local/Remote mode
	        IF #QREMOTE=false THEN
	          // Local mode is active
	          // OPEN/CLOSE valve by linking (MAN_OP)
	          #QCMD_OP:=#MAN_OP AND NOT #QMAN_AUT;
	          #OPdwCmd.%X0:=false;
	          #OPdwCmd.%X1:=false;
	        ELSE
	         // Remote mode is active
	          // Open valve by operator
	          IF #OPdwCmd.%X1=true THEN
	            #QCMD_OP:=true;
	            #OPdwCmd.%X0:=false;
	            #OPdwCmd.%X1:=false;
	          END_IF;
	          // Close valve by operator
	          IF #OPdwCmd.%X0=true THEN
	            #QCMD_OP:=false;
	            #OPdwCmd.%X0:=false;
	            #OPdwCmd.%X1:=false;
	          END_IF;
	        END_IF;
	      END_IF;
	    ELSE
	      // Local/Remote mode
	      IF #QREMOTE=false THEN
	        // Local mode is active
	          // OPEN/CLOSE valve by linking (SIM_OP)
	          #QCMD_SIM:=#SIM_OP;
	          #OPdwCmd.%X0:=false;
	          #OPdwCmd.%X1:=false;
	      ELSE
	        // Remote mode is active
	          // Open valve by operator
	          IF #OPdwCmd.%X1=true THEN
	            #QCMD_SIM:=true;
	            #OPdwCmd.%X0:=false;
	            #OPdwCmd.%X1:=false;
	          END_IF;
	          // Close valve by operator
	          IF #OPdwCmd.%X0=true THEN
	            #QCMD_SIM:=false;
	            #OPdwCmd.%X0:=false;
	            #OPdwCmd.%X1:=false;
	          END_IF;        
	        END_IF;    
	    END_IF;  
	  ELSE
	    // Errors occurs
	    #QCMD_OP:=false;
	    #QCMD_SIM:=false;
	  END_IF;
	
	  (****************************************
	    Network 7: Control signal to the valve
	  *****************************************)
	  IF #QERR=false THEN
	    // Close  valve
	    IF (((#FB_CLOSE=true OR #QMON=false) AND #QSIM=false AND #QCMD_OP=false) OR
	      ((#FB_SIM_CLOSE=true OR #QMON=false) AND #QSIM=true AND #QCMD_SIM=false)) AND #QCLOSING=true THEN
	      #QCLOSE:=true;
	      #QCLOSING:=false;
	      #QOPEN:=false;
	      #QOPENING:=false;
	      #QwState := 0;
	    END_IF;
	    // Closing valve
	    IF ((#QSIM=false AND #QCMD_OP=false) OR (#QSIM=true AND #QCMD_SIM=false)) AND (#QOPEN=true OR #QOPENING=true) THEN
	      #QCLOSE:=false;
	      #QCLOSING:=true;
	      #QOPEN:=false;
	      #QOPENING:=false;
	      #QwState := 3;
	    END_IF;
	    // Open valve
	    IF (((#FB_OPEN=true OR #QMON=false) AND #QSIM=false AND #QCMD_OP=true) OR
	      ((#FB_SIM_OPEN=true OR #QMON=false) AND #QSIM=true AND #QCMD_SIM=true)) AND #QOPENING=true THEN    
	    #QCLOSE:=false;
	    #QCLOSING:=false;
	    #QOPEN:=true;
	    #QOPENING:=false;
	    #QwState := 2;
	    END_IF;
	    // Opening valve
	    IF ((#QSIM=false AND #QCMD_OP=true) OR (#QSIM=true AND #QCMD_SIM=true)) AND (#QCLOSE=true OR #QCLOSING=true) THEN
	    #QCLOSE:=false;
	    #QCLOSING:=false;
	    #QOPEN:=false;
	    #QOPENING:=true;
	    #QwState := 1;
	    END_IF;
	  END_IF;
	
	  (*******************************************************************
	    Network 8: Feedbacks for monitoring in process and simulation mode
	  ********************************************************************)
	  IF #QSIM=false AND #QMON=true  THEN
	  // Feedback monitoring in process mode
	    #TOPENING(IN:=#QOPENING,
	               PT:=#MON_T,
	               Q=>#MON_ERR_OPENING,
	               ET=>#QMON_T);
	     
	    #TCLOSING(IN:=#QCLOSING,
	              PT:=#MON_T_CLOSE,
	              Q=>#MON_ERR_CLOSING,
	              ET=>#QMON_T_CLOSE);
	    // Feedback error
	    #FB_ERR:= ((NOT #FB_OPEN OR #FB_CLOSE) AND #QOPEN) OR ((#FB_OPEN OR NOT #FB_CLOSE) AND #QCLOSE);
	    IF #FB_ERR=true OR #MON_ERR_OPENING=true OR #MON_ERR_CLOSING=true THEN
	      #QMON_ERR:=true;
	    END_IF;
	    
	    
	  ELSIF #QSIM=true AND #QMON=true THEN
	    // Feedback monitoring in simulation mode
	    #TOPENING_SIM(IN:=#QOPENING,
	                  PT:=#SIM_T,
	                  Q=>#MON_SIM_OPENING,
	                  ET=>#QSIM_T);
	    
	    #TCLOSING_SIM(IN:=#QCLOSING,
	                  PT:=#SIM_T_CLOSE,
	                  Q=>#MON_SIM_CLOSING,
	                  ET=>#QSIM_T_CLOSE);
	    
	    // Feedback for open in simulation mode
	    IF #MON_SIM_CLOSING=true OR #QERR=true THEN
	      #FB_SIM_OPEN:=false;
	    ELSIF #MON_SIM_OPENING=true THEN
	      #FB_SIM_OPEN:=true;
	    END_IF;
	     // Feedback for close in simulation mode
	    #FB_SIM_CLOSE:=NOT #FB_SIM_OPEN;
	  END_IF;
	  
	  (**********************************************
	    Network 9: Check errors
	  ***********************************************)
	  // External error
	  #QERR_EXT:=#ERR_EXTERN;  
	  // Interlock error
	  IF #LOCK=true AND ( #QOPEN=true OR #QOPENING=true) THEN
	    #QLOCK:=true;
	  END_IF;
	  // Error in valve condition
	  #CON_ERR:=NOT((#QCLOSE AND NOT #QCLOSING AND NOT #QOPENING AND NOT #QOPEN) OR
	  (NOT #QCLOSE AND #QCLOSING AND NOT #QOPENING AND NOT #QOPEN) OR
	  (NOT #QCLOSE AND NOT #QCLOSING AND  #QOPENING AND NOT #QOPEN) OR
	  (NOT #QCLOSE AND NOT #QCLOSING AND NOT #QOPENING AND  #QOPEN));
	
	  (**********************************************
	    Network 10: General error
	  ***********************************************)
	  #QERR:= #QERR_EXT OR #QMON_ERR OR #QLOCK OR #CON_ERR;
	
	  (**********************************************
	    Network 11: If error then stop
	  ***********************************************)
	  IF #QERR=true THEN
	    #QCLOSE:=true;
	    #QCLOSING:=false;
	    #QOPEN:=false;
	    #QOPENING:=false;
	    #QwState := 0;
	  END_IF;
	
	  IF #OP_RESET=true THEN
	    #QMON_ERR:=false;
	    #QLOCK:=false;
	  END_IF;
	  
	  // End normal case
	END_IF;
	
	(****************************************************
	  Network 1: Influence visibility of faceplate window
	*****************************************************)
	IF #OP_VISIBILITY<>#VISIBILITY_OLD THEN
	  #VISIBILITY_OLD:=#OP_VISIBILITY;
	  #VISIBILITY:=#OP_VISIBILITY;
	ELSIF #VISIBILITY<>#VISIBILITY_OLD THEN
	  #VISIBILITY_OLD:=#VISIBILITY;
	  #OP_VISIBILITY:=#VISIBILITY;
	END_IF;
	(********************************
	  Network 10: Set state for HMI
	*********************************)
	#QdwState.%X0:=#QCLOSE AND NOT #QERR;
	#QdwState.%X1:=#QOPENING;
	#QdwState.%X2:=#QOPEN;
	#QdwState.%X3:=#QCLOSING;
	#QdwState.%X4:=false;
	#QdwState.%X5:=false;
	#QdwState.%X6:=false;
	#QdwState.%X7:=false;
	#QdwState.%X8:=#QMON;
	#QdwState.%X9:=#QMON_ERR;
	#QdwState.%X10:=false;
	#QdwState.%X11:=false;
	#QdwState.%X12:=false;
	#QdwState.%X13:=false;
	#QdwState.%X14:=false;
	#QdwState.%X15:=false;
	#QdwState.%X16:=#QMAN_AUT;
	#QdwState.%X17:=#QREMOTE;
	#QdwState.%X18:=#QSIM;
	#QdwState.%X19:=false;
	#QdwState.%X20:=false;
	#QdwState.%X21:=false;
	#QdwState.%X22:=false;
	#QdwState.%X23:=false;
	#QdwState.%X24:=#QERR;
	#QdwState.%X25:=#QERR_EXT;
	#QdwState.%X26:=#QLOCK;
	#QdwState.%X27:=#LOCK;
	#QdwState.%X28:=false;
	#QdwState.%X29:=false;
	#QdwState.%X30:=false;
	#QdwState.%X31:=false;
	
	(********************************
	  Network 11: Bit alarm procedure
	*********************************)
	#QwAlarm.%X0:=#QMON_ERR;
	#QwAlarm.%X1:=false;
	#QwAlarm.%X2:=false;
	#QwAlarm.%X3:=false;
	#QwAlarm.%X4:=#QLOCK;
	#QwAlarm.%X5:=false;
	#QwAlarm.%X6:=#QERR_EXT;
	#QwAlarm.%X7:=#QERR;
	#QwAlarm.%X8:=#QCLOSE;
	#QwAlarm.%X9:=#QOPENING;
	#QwAlarm.%X10:=#QOPEN;
	#QwAlarm.%X11:=#QCLOSING;
	#QwAlarm.%X12:=#LOCK;
	#QwAlarm.%X13:=#QREMOTE;
	#QwAlarm.%X14:=#QMAN_AUT;
	#QwAlarm.%X15:=#QSIM;
END_FUNCTION_BLOCK

FUNCTION_BLOCK "IO Valve T03 Chili"   // FB303, LAD
{ S7_Optimized_Access := 'FALSE' }
VERSION : 0.1
// stored: AutoNumber false, IsIECCheckEnabled false, SetENOAutomatically false, UDAEnableTagReadback false
   VAR_INPUT
      lock : Bool;
      Init : Bool;
      testing : Bool;
      Reset : Bool;
   END_VAR
   VAR
      "AV-03.01" { S7_SetPoint := 'True'} : "Valve";   // AUTO BUTTERFLY VALVE INLET PROCESS WATER TO BFT CHILI AWETAN T-03.00
      "AV-03.02" { S7_SetPoint := 'True'} : "Valve";   // AUTO BUTTERFLY VALVE CIP SUPPLY TO BFT CHILI AWETAN T-03.00
      "AV-03.03" { S7_SetPoint := 'True'} : "Valve";   // AUTO BUTTERFLY VALVE OUTLET PRODUCT FROM BFT CHILI AWETAN T-03.00
      "AV-03.04" { S7_SetPoint := 'True'} : "Valve";   // AUTO BUTTERFLY VALVE OUTLET CIP TANK & LINE CHILI AWETAN T-03.00
      "AV-03.05" { S7_SetPoint := 'True'} : "Valve";   // AUTO BUTTERFLY VALVE DRAIN MONO PUMP P-03.01
      "AV-03.06" { S7_SetPoint := 'True'} : "Valve";   // AUTO BUTTERFLY VALVE INLET PRODUCT TO BFT CHILI AWETAN T-03.00
      "AV-03.07" { S7_SetPoint := 'True'} : "Valve";   // AUTO BUTTERFLY VALVE INLET CHILI AWETAN FROM T-02.00 TO BLENDING TANK T-20.00
      "AV-03.08" { S7_SetPoint := 'True'} : "Valve";
      "AV-03.09" { S7_SetPoint := 'True'} : "Valve";
      "AV-03.10" { S7_SetPoint := 'True'} : "Valve";
      "AV-03.11" { S7_SetPoint := 'True'} : "Valve";
      "AV-03.12" { S7_SetPoint := 'True'} : "Valve";
      "AV-03.13" { S7_SetPoint := 'True'} : "Valve";
      "AV-03.14" { S7_SetPoint := 'True'} : "Valve";
      "AV-03.15" { S7_SetPoint := 'True'} : "Valve";
   END_VAR
BEGIN

REGION Network 1 (SCL): FB OPEN and CLOSE
   IF #testing THEN
       // Statement section IF
       #"AV-03.01".FB_OPEN := #"AV-03.01".QCMD_OP;
       #"AV-03.01".FB_CLOSE := NOT #"AV-03.01".QCMD_OP;
       #"AV-03.02".FB_OPEN := #"AV-03.02".QCMD_OP;
       #"AV-03.02".FB_CLOSE := NOT #"AV-03.02".QCMD_OP;
       #"AV-03.03".FB_OPEN := #"AV-03.03".QCMD_OP;
       #"AV-03.03".FB_CLOSE := NOT #"AV-03.03".QCMD_OP;
       #"AV-03.04".FB_OPEN := #"AV-03.04".QCMD_OP;
       #"AV-03.04".FB_CLOSE := NOT #"AV-03.04".QCMD_OP;
       #"AV-03.05".FB_OPEN := #"AV-03.05".QCMD_OP;
       #"AV-03.05".FB_CLOSE := NOT #"AV-03.05".QCMD_OP;
       #"AV-03.06".FB_OPEN := #"AV-03.06".QCMD_OP;
       #"AV-03.06".FB_CLOSE := NOT #"AV-03.06".QCMD_OP;
       #"AV-03.07".FB_OPEN := #"AV-03.07".QCMD_OP;
       #"AV-03.07".FB_CLOSE := NOT #"AV-03.07".QCMD_OP;
       #"AV-03.08".FB_OPEN := #"AV-03.08".QCMD_OP;
       #"AV-03.08".FB_CLOSE := NOT #"AV-03.08".QCMD_OP;
       #"AV-03.09".FB_OPEN := #"AV-03.09".QCMD_OP;
       #"AV-03.09".FB_CLOSE := NOT #"AV-03.09".QCMD_OP;
       #"AV-03.10".FB_OPEN := #"AV-03.10".QCMD_OP;
       #"AV-03.10".FB_CLOSE := NOT #"AV-03.10".QCMD_OP;
       #"AV-03.11".FB_OPEN := #"AV-03.11".QCMD_OP;
       #"AV-03.11".FB_CLOSE := NOT #"AV-03.11".QCMD_OP;
       #"AV-03.12".FB_OPEN := #"AV-03.12".QCMD_OP;
       #"AV-03.12".FB_CLOSE := NOT #"AV-03.12".QCMD_OP;
       #"AV-03.13".FB_OPEN := #"AV-03.13".QCMD_OP;
       #"AV-03.13".FB_CLOSE := NOT #"AV-03.13".QCMD_OP;
       #"AV-03.14".FB_OPEN := #"AV-03.14".QCMD_OP;
       #"AV-03.14".FB_CLOSE := NOT #"AV-03.14".QCMD_OP;
       #"AV-03.15".FB_OPEN := #"AV-03.15".QCMD_OP;
       #"AV-03.15".FB_CLOSE := NOT #"AV-03.15".QCMD_OP;
   ELSE
       // Statement section ELSE
       #"AV-03.01".FB_OPEN := NOT "ZSC-03.01";
       #"AV-03.01".FB_CLOSE := "ZSC-03.01";
       #"AV-03.02".FB_OPEN := NOT "ZSC-03.02";
       #"AV-03.02".FB_CLOSE := "ZSC-03.02";
       #"AV-03.03".FB_OPEN := NOT "ZSC-03.03";
       #"AV-03.03".FB_CLOSE := "ZSC-03.03";
       #"AV-03.04".FB_OPEN := NOT "ZSC-03.04";
       #"AV-03.04".FB_CLOSE := "ZSC-03.04";
       #"AV-03.05".FB_OPEN := #"AV-03.05".QCMD_OP;
       #"AV-03.05".FB_CLOSE := NOT #"AV-03.05".QCMD_OP;
       #"AV-03.06".FB_OPEN := NOT "ZSC-03.06";
       #"AV-03.06".FB_CLOSE := "ZSC-03.06";
       #"AV-03.07".FB_OPEN := #"AV-03.07".QCMD_OP;
       #"AV-03.07".FB_CLOSE := NOT #"AV-03.07".QCMD_OP;
       #"AV-03.08".FB_OPEN := #"AV-03.08".QCMD_OP;
       #"AV-03.08".FB_CLOSE := NOT #"AV-03.08".QCMD_OP;
       #"AV-03.09".FB_OPEN := #"AV-03.09".QCMD_OP;
       #"AV-03.09".FB_CLOSE := NOT #"AV-03.09".QCMD_OP;
       #"AV-03.10".FB_OPEN := #"AV-03.10".QCMD_OP;
       #"AV-03.10".FB_CLOSE := NOT #"AV-03.10".QCMD_OP;
       #"AV-03.11".FB_OPEN := NOT "ZSC-03.11";
       #"AV-03.11".FB_CLOSE := "ZSC-03.11";
       #"AV-03.12".FB_OPEN := NOT "ZSC-03.12";
       #"AV-03.12".FB_CLOSE := "ZSC-03.12";
       #"AV-03.13".FB_OPEN := NOT "ZSC-03.13";
       #"AV-03.13".FB_CLOSE := "ZSC-03.13";
       #"AV-03.14".FB_OPEN := #"AV-03.14".QCMD_OP;
       #"AV-03.14".FB_CLOSE := NOT #"AV-03.14".QCMD_OP;
       #"AV-03.15".FB_OPEN := #"AV-03.15".QCMD_OP;
       #"AV-03.15".FB_CLOSE := NOT #"AV-03.15".QCMD_OP;
   END_IF;
END_REGION

